C03641=1096.665,388.790,405.608,178.895,21.471,152.910
C03642=1096.660,388.542,405.645,178.892,21.465,152.909
C03643=1096.654,388.296,405.683,178.889,21.458,152.908
C03644=1096.648,388.049,405.721,178.886,21.452,152.907
C03645=1096.642,387.801,405.758,178.884,21.446,152.906
C03646=1096.637,387.555,405.796,178.881,21.440,152.905
C03647=1096.631,387.308,405.834,178.878,21.434,152.904
C03648=1096.625,387.061,405.871,178.876,21.428,152.903
C03649=1096.619,386.814,405.908,178.873,21.422,152.902
C03650=1096.614,386.567,405.945,178.869,21.416,152.901
C03651=1096.608,386.320,405.983,178.867,21.410,152.900
C03652=1096.601,386.072,406.021,178.864,21.404,152.899
C03653=1096.595,385.825,406.058,178.861,21.398,152.898
C03654=1096.590,385.579,406.094,178.859,21.392,152.897
C03655=1096.583,385.331,406.132,178.856,21.387,152.896
C03656=1096.578,385.084,406.170,178.853,21.381,152.895
C03657=1096.573,384.837,406.206,178.851,21.375,152.894
C03658=1096.567,384.590,406.244,178.847,21.369,152.893
C03659=1096.561,384.378,406.276,178.845,21.364,152.892
C03660=1096.556,384.167,406.308,178.843,21.359,152.891
C03661=1096.552,383.955,406.339,178.840,21.354,152.890
C03662=1096.546,383.743,406.371,178.838,21.349,152.890
C03663=1096.541,383.532,406.403,178.836,21.344,152.889
C03664=1096.536,383.321,406.435,178.833,21.339,152.888
C03665=1096.532,383.109,406.467,178.831,21.334,152.887
C03666=1096.527,382.897,406.499,178.828,21.329,152.886
C03667=1096.521,382.650,406.535,178.826,21.324,152.885
C03668=1096.515,382.403,406.572,178.823,21.318,152.885
C03669=1096.510,382.156,406.610,178.819,21.312,152.884
C03670=1096.503,381.909,406.646,178.816,21.306,152.883
C03671=1096.498,381.662,406.683,178.814,21.301,152.882
C03672=1096.492,381.414,406.720,178.811,21.295,152.881
C03673=1096.486,381.167,406.757,178.808,21.289,152.880
C03674=1096.480,380.920,406.794,178.805,21.284,152.879
C03675=1096.473,380.674,406.831,178.802,21.279,152.878
C03676=1096.468,380.426,406.868,178.799,21.273,152.877
C03677=1096.462,380.179,406.905,178.797,21.267,152.876
C03678=1096.456,379.932,406.942,178.794,21.262,152.876
C03679=1096.450,379.684,406.979,178.791,21.256,152.875
C03680=1096.445,379.438,407.015,178.788,21.251,152.874
C03681=1096.439,379.191,407.052,178.785,21.246,152.873
C03682=1096.433,378.944,407.088,178.782,21.240,152.872
C03683=1096.427,378.696,407.125,178.780,21.234,152.871
C03684=1096.421,378.449,407.162,178.777,21.229,152.870
C03685=1096.415,378.202,407.199,178.774,21.223,152.870
C03686=1096.410,377.955,407.236,178.771,21.218,152.869
C03687=1096.404,377.708,407.271,178.768,21.213,152.868
C03688=1096.398,377.460,407.308,178.765,21.207,152.867
C03689=1096.392,377.213,407.345,178.762,21.202,152.866
C03690=1096.387,376.966,407.382,178.759,21.196,152.865
C03691=1096.380,376.719,407.418,178.756,21.191,152.865
C03692=1096.375,376.472,407.455,178.754,21.186,152.864
C03693=1096.369,376.224,407.491,178.751,21.181,152.863
C03694=1096.364,375.977,407.528,178.748,21.176,152.862
C03695=1096.357,375.730,407.564,178.746,21.170,152.861
C03696=1096.352,375.483,407.601,178.743,21.165,152.860
C03697=1096.346,375.236,407.636,178.740,21.159,152.860
C03698=1096.341,374.988,407.673,178.737,21.154,152.859
C03699=1096.334,374.741,407.710,178.734,21.149,152.858
C03700=1096.329,374.494,407.745,178.731,21.144,152.857
C03701=1096.323,374.247,407.782,178.728,21.138,152.856
C03702=1096.317,374.000,407.819,178.725,21.133,152.856
C03703=1096.311,373.752,407.854,178.722,21.128,152.855
C03704=1096.305,373.505,407.892,178.719,21.123,152.854
C03705=1096.300,373.258,407.927,178.717,21.118,152.853
C03706=1096.294,373.011,407.963,178.714,21.113,152.853
C03707=1096.288,372.763,407.999,178.711,21.108,152.852
C03708=1096.282,372.516,408.036,178.708,21.102,152.851
C03709=1096.276,372.269,408.071,178.705,21.098,152.850
C03710=1096.270,372.022,408.108,178.702,21.092,152.850
C03711=1096.264,371.774,408.144,178.699,21.087,152.849
C03712=1096.259,371.527,408.181,178.696,21.082,152.848
C03713=1096.253,371.280,408.216,178.693,21.078,152.847
C03714=1096.247,371.033,408.252,178.691,21.072,152.847
C03715=1096.237,370.636,408.310,178.686,21.064,152.845
C03716=1096.228,370.241,408.368,178.681,21.056,152.844
C03717=1096.218,369.845,408.425,178.676,21.048,152.843
C03718=1096.210,369.448,408.483,178.672,21.041,152.842
C03719=1096.204,369.201,408.518,178.669,21.036,152.841
C03720=1096.198,368.954,408.555,178.666,21.031,152.841
C03721=1096.192,368.707,408.590,178.663,21.026,152.840
C03722=1096.187,368.460,408.626,178.659,21.021,152.839
C03723=1096.181,368.212,408.661,178.656,21.016,152.838
C03724=1096.175,367.965,408.698,178.654,21.011,152.838
C03725=1096.170,367.718,408.734,178.651,21.007,152.837
C03726=1096.164,367.470,408.770,178.648,21.001,152.836
C03727=1096.158,367.223,408.805,178.645,20.997,152.836
C03728=1096.152,366.975,408.841,178.642,20.992,152.835
C03729=1096.146,366.728,408.876,178.640,20.987,152.834
C03730=1096.141,366.481,408.912,178.636,20.982,152.834
C03731=1096.134,366.234,408.948,178.633,20.977,152.833
C03732=1096.129,365.987,408.984,178.630,20.973,152.832
C03733=1096.123,365.739,409.019,178.627,20.967,152.832
C03734=1096.118,365.492,409.055,178.625,20.963,152.831
C03735=1096.111,365.244,409.090,178.622,20.958,152.830
C03736=1096.105,364.997,409.126,178.619,20.953,152.830
C03737=1096.100,364.750,409.161,178.615,20.949,152.829
C03738=1096.094,364.502,409.197,178.612,20.944,152.828
C03739=1096.089,364.255,409.232,178.610,20.939,152.828
C03740=1096.083,364.007,409.268,178.607,20.935,152.827
C03741=1096.077,363.760,409.303,178.603,20.930,152.827
C03742=1096.071,363.512,409.339,178.600,20.925,152.826
C03743=1096.065,363.266,409.373,178.598,20.921,152.825
C03744=1096.059,363.018,409.409,178.595,20.916,152.825
C03745=1096.053,362.770,409.445,178.592,20.912,152.824
C03746=1096.048,362.523,409.480,178.588,20.907,152.824
C03747=1096.042,362.275,409.515,178.586,20.903,152.823
C03748=1096.037,362.028,409.551,178.583,20.898,152.822
C03749=1096.031,361.780,409.586,178.580,20.893,152.822
C03750=1096.024,361.534,409.621,178.577,20.889,152.821
C03751=1096.019,361.285,409.656,178.574,20.885,152.821
C03752=1096.013,361.038,409.691,178.571,20.880,152.820
C03753=1096.008,360.791,409.727,178.567,20.875,152.819
C03754=1096.002,360.544,409.763,178.565,20.871,152.819
C03755=1095.996,360.296,409.797,178.562,20.866,152.818
C03756=1095.990,360.049,409.832,178.559,20.862,152.818
C03757=1095.985,359.801,409.867,178.556,20.858,152.817
C03758=1095.979,359.553,409.903,178.553,20.853,152.817
C03759=1095.973,359.307,409.937,178.550,20.848,152.816
C03760=1095.967,359.059,409.973,178.546,20.844,152.815
C03761=1095.961,358.812,410.008,178.544,20.840,152.815
C03762=1095.955,358.564,410.042,178.541,20.835,152.814
C03763=1095.950,358.317,410.078,178.537,20.831,152.814
C03764=1095.944,358.069,410.112,178.535,20.827,152.813
C03765=1095.938,357.822,410.147,178.532,20.822,152.813
C03766=1095.933,357.574,410.182,178.528,20.818,152.812
C03767=1095.923,357.194,410.236,178.524,20.811,152.811
C03768=1095.914,356.813,410.290,178.520,20.804,152.810
C03769=1095.906,356.432,410.344,178.515,20.798,152.810
C03770=1095.897,356.051,410.397,178.511,20.791,152.809
C03771=1095.891,355.803,410.432,178.507,20.787,152.808
C03772=1095.885,355.556,410.466,178.504,20.782,152.808
C03773=1095.880,355.309,410.501,178.501,20.779,152.807
C03774=1095.873,355.061,410.536,178.498,20.774,152.807
C03775=1095.868,354.814,410.571,178.495,20.769,152.806
C03776=1095.862,354.566,410.605,178.492,20.765,152.806
C03777=1095.856,354.318,410.640,178.489,20.761,152.805
C03778=1095.851,354.071,410.675,178.487,20.757,152.805
C03779=1095.845,353.824,410.709,178.483,20.753,152.804
C03780=1095.839,353.576,410.744,178.480,20.748,152.804
C03781=1095.833,353.328,410.778,178.477,20.745,152.803
C03782=1095.828,353.081,410.813,178.474,20.740,152.803
C03783=1095.822,352.833,410.847,178.471,20.736,152.802
C03784=1095.816,352.586,410.882,178.468,20.732,152.802
C03785=1095.810,352.338,410.917,178.465,20.728,152.801
C03786=1095.805,352.091,410.951,178.462,20.724,152.801
C03787=1095.798,351.843,410.985,178.459,20.720,152.800
C03788=1095.793,351.596,411.020,178.455,20.715,152.800
C03789=1095.787,351.348,411.054,178.453,20.711,152.799
C03790=1095.781,351.100,411.089,178.450,20.707,152.799
C03791=1095.776,350.853,411.123,178.447,20.704,152.798
C03792=1095.770,350.605,411.157,178.443,20.699,152.798
C03793=1095.765,350.358,411.192,178.440,20.695,152.797
C03794=1095.758,350.110,411.226,178.438,20.691,152.797
C03795=1095.752,349.863,411.260,178.434,20.687,152.797
C03796=1095.747,349.615,411.295,178.432,20.683,152.796
C03797=1095.741,349.368,411.329,178.428,20.679,152.796
C03798=1095.735,349.120,411.363,178.425,20.675,152.795
C03799=1095.730,348.872,411.398,178.422,20.671,152.795
C03800=1095.724,348.625,411.432,178.420,20.667,152.794
C03801=1095.718,348.377,411.466,178.416,20.663,152.794
C03802=1095.712,348.130,411.500,178.413,20.659,152.793
C03803=1095.707,347.881,411.535,178.410,20.655,152.793
C03804=1095.701,347.634,411.569,178.407,20.651,152.793
C03805=1095.695,347.387,411.603,178.404,20.647,152.792
C03806=1095.689,347.140,411.637,178.401,20.643,152.792
C03807=1095.684,346.891,411.671,178.398,20.639,152.791
C03808=1095.678,346.644,411.705,178.395,20.635,152.791
C03809=1095.672,346.396,411.739,178.392,20.631,152.790
C03810=1095.666,346.148,411.772,178.389,20.627,152.790
C03811=1095.661,345.901,411.807,178.386,20.624,152.790
C03812=1095.655,345.654,411.841,178.382,20.619,152.789
C03813=1095.650,345.406,411.875,178.380,20.616,152.789
C03814=1095.644,345.158,411.909,178.376,20.612,152.788
C03815=1095.638,344.911,411.943,178.373,20.608,152.788
C03816=1095.633,344.663,411.976,178.370,20.604,152.788
C03817=1095.626,344.415,412.010,178.367,20.600,152.787
C03818=1095.620,344.168,412.044,178.364,20.596,152.787
C03819=1095.612,343.789,412.096,178.359,20.590,152.786
C03820=1095.603,343.411,412.147,178.355,20.584,152.786
C03821=1095.594,343.032,412.199,178.350,20.579,152.785
C03822=1095.586,342.654,412.250,178.346,20.574,152.784
C03823=1095.580,342.406,412.285,178.342,20.569,152.784
C03824=1095.574,342.158,412.318,178.340,20.566,152.784
C03825=1095.568,341.911,412.352,178.336,20.562,152.783
C03826=1095.563,341.663,412.385,178.333,20.558,152.783
C03827=1095.557,341.416,412.419,178.330,20.554,152.783
C03828=1095.551,341.168,412.452,178.327,20.551,152.782
C03829=1095.545,340.920,412.485,178.323,20.547,152.782
C03830=1095.539,340.673,412.519,178.321,20.544,152.782
C03831=1095.534,340.425,412.553,178.317,20.540,152.781
C03832=1095.528,340.177,412.586,178.314,20.536,152.781
C03833=1095.522,339.930,412.620,178.311,20.532,152.780
C03834=1095.517,339.682,412.654,178.308,20.529,152.780
C03835=1095.511,339.434,412.687,178.306,20.525,152.780
C03836=1095.505,339.187,412.721,178.302,20.521,152.779
C03837=1095.500,338.939,412.754,178.300,20.517,152.779
C03838=1095.494,338.691,412.788,178.296,20.514,152.779
C03839=1095.486,338.352,412.833,178.292,20.509,152.778
C03840=1095.479,338.012,412.879,178.287,20.504,152.778
C03841=1095.469,337.673,412.925,178.283,20.499,152.777
C03842=1095.462,337.333,412.971,178.279,20.494,152.777
C03843=1095.456,337.085,413.004,178.276,20.491,152.776
C03844=1095.450,336.838,413.037,178.273,20.487,152.776
C03845=1095.445,336.590,413.070,178.270,20.484,152.776
C03846=1095.439,336.342,413.104,178.266,20.480,152.776
C03847=1095.434,336.095,413.137,178.264,20.476,152.775
C03848=1095.428,335.847,413.169,178.261,20.473,152.775
C03849=1095.422,335.599,413.203,178.257,20.469,152.775
C03850=1095.417,335.351,413.236,178.254,20.466,152.774
C03851=1095.410,335.104,413.269,178.251,20.462,152.774
C03852=1095.405,334.856,413.302,178.248,20.459,152.774
C03853=1095.399,334.608,413.335,178.245,20.455,152.773
C03854=1095.394,334.360,413.369,178.242,20.451,152.773
C03855=1095.387,334.112,413.402,178.239,20.448,152.773
C03856=1095.382,333.864,413.435,178.236,20.445,152.772
C03857=1095.376,333.617,413.468,178.233,20.441,152.772
C03858=1095.371,333.370,413.501,178.230,20.438,152.772
C03859=1095.365,333.122,413.534,178.226,20.434,152.772
C03860=1095.359,332.874,413.567,178.223,20.431,152.771
C03861=1095.353,332.626,413.599,178.221,20.427,152.771
C03862=1095.348,332.378,413.633,178.217,20.424,152.771
C03863=1095.342,332.130,413.665,178.214,20.421,152.770
C03864=1095.336,331.882,413.699,178.211,20.417,152.770
C03865=1095.330,331.635,413.731,178.208,20.414,152.770
C03866=1095.325,331.387,413.764,178.205,20.411,152.770
C03867=1095.319,331.139,413.796,178.202,20.407,152.769
C03868=1095.313,330.891,413.830,178.198,20.404,152.769
C03869=1095.307,330.644,413.863,178.195,20.401,152.769
C03870=1095.301,330.396,413.895,178.193,20.397,152.769
C03871=1095.295,330.104,413.934,178.189,20.394,152.768
C03872=1095.287,329.811,413.973,178.184,20.389,152.768
C03873=1095.281,329.518,414.011,178.181,20.385,152.768
C03874=1095.273,329.226,414.049,178.177,20.381,152.767
C03875=1095.268,328.978,414.083,178.175,20.378,152.767
C03876=1095.262,328.729,414.115,178.172,20.375,152.767
C03877=1095.256,328.483,414.147,178.168,20.371,152.767
C03878=1095.251,328.234,414.180,178.165,20.368,152.767
C03879=1095.245,327.986,414.212,178.162,20.365,152.766
C03880=1095.238,327.739,414.245,178.158,20.361,152.766
C03881=1095.233,327.490,414.278,178.156,20.358,152.766
C03882=1095.227,327.243,414.310,178.153,20.355,152.766
C03883=1095.221,326.995,414.342,178.150,20.352,152.765
C03884=1095.216,326.747,414.375,178.146,20.348,152.765
C03885=1095.210,326.499,414.407,178.143,20.345,152.765
C03886=1095.204,326.252,414.440,178.140,20.342,152.765
C03887=1095.199,326.004,414.472,178.137,20.339,152.764
C03888=1095.193,325.755,414.505,178.134,20.336,152.764
C03889=1095.187,325.508,414.537,178.131,20.333,152.764
C03890=1095.181,325.260,414.569,178.128,20.329,152.764
C03891=1095.176,325.012,414.602,178.124,20.326,152.763
C03892=1095.170,324.764,414.634,178.121,20.323,152.763
C03893=1095.164,324.517,414.666,178.118,20.320,152.763
C03894=1095.158,324.269,414.699,178.115,20.316,152.763
C03895=1095.153,324.021,414.731,178.112,20.313,152.763
C03896=1095.147,323.773,414.763,178.109,20.310,152.762
C03897=1095.141,323.525,414.796,178.106,20.307,152.762
C03898=1095.135,323.277,414.828,178.102,20.304,152.762
C03899=1095.130,323.030,414.859,178.099,20.301,152.762
C03900=1095.125,322.781,414.892,178.096,20.298,152.762
C03901=1095.118,322.534,414.925,178.094,20.295,152.761
C03902=1095.113,322.286,414.956,178.090,20.291,152.761
C03903=1095.107,322.038,414.988,178.087,20.288,152.761
C03904=1095.101,321.790,415.020,178.084,20.285,152.761
C03905=1095.096,321.543,415.053,178.081,20.282,152.761
C03906=1095.090,321.294,415.085,178.078,20.279,152.760
C03907=1095.085,321.047,415.117,178.074,20.275,152.760
C03908=1095.079,320.799,415.149,178.071,20.272,152.760
C03909=1095.073,320.551,415.181,178.069,20.269,152.760
C03910=1095.067,320.303,415.213,178.066,20.266,152.759
C03911=1095.063,320.055,415.245,178.062,20.263,152.759
C03912=1095.057,319.807,415.277,178.059,20.260,152.759
C03913=1095.051,319.559,415.309,178.056,20.257,152.759
C03914=1095.045,319.311,415.341,178.053,20.254,152.759
C03915=1095.039,319.063,415.373,178.050,20.251,152.758
C03916=1095.034,318.815,415.405,178.046,20.247,152.758
C03917=1095.028,318.567,415.437,178.044,20.244,152.758
C03918=1095.022,318.320,415.468,178.041,20.241,152.758
C03919=1095.016,318.071,415.500,178.038,20.238,152.758
C03920=1095.011,317.824,415.532,178.034,20.235,152.757
C03921=1095.006,317.575,415.565,178.031,20.232,152.757
C03922=1095.000,317.328,415.596,178.028,20.229,152.757
C03923=1094.992,316.937,415.646,178.023,20.224,152.757
C03924=1094.982,316.546,415.696,178.018,20.219,152.757
C03925=1094.973,316.154,415.746,178.013,20.214,152.756
C03926=1094.965,315.762,415.796,178.009,20.210,152.756
C03927=1094.959,315.515,415.828,178.005,20.206,152.756
C03928=1094.954,315.267,415.860,178.002,20.203,152.756
C03929=1094.948,315.019,415.892,177.999,20.201,152.755
C03930=1094.942,314.770,415.923,177.996,20.198,152.755
C03931=1094.936,314.523,415.954,177.993,20.195,152.755
C03932=1094.930,314.275,415.986,177.990,20.192,152.755
C03933=1094.925,314.027,416.018,177.986,20.189,152.755
C03934=1094.919,313.779,416.049,177.983,20.186,152.755
C03935=1094.913,313.531,416.080,177.980,20.183,152.755
C03936=1094.907,313.283,416.112,177.977,20.180,152.754
C03937=1094.902,313.036,416.144,177.974,20.178,152.754
C03938=1094.896,312.788,416.174,177.971,20.175,152.754
C03939=1094.890,312.540,416.206,177.968,20.172,152.754
C03940=1094.884,312.292,416.238,177.964,20.169,152.754
C03941=1094.878,312.044,416.269,177.961,20.166,152.754
C03942=1094.873,311.796,416.300,177.958,20.163,152.754
C03943=1094.867,311.547,416.332,177.955,20.161,152.754
C03944=1094.861,311.300,416.363,177.952,20.158,152.754
C03945=1094.856,311.052,416.394,177.949,20.155,152.753
C03946=1094.849,310.804,416.425,177.946,20.152,152.753
C03947=1094.844,310.557,416.457,177.942,20.149,152.753
C03948=1094.838,310.308,416.488,177.939,20.146,152.753
C03949=1094.832,310.061,416.519,177.936,20.143,152.753
C03950=1094.827,309.812,416.550,177.933,20.141,152.753
C03951=1094.821,309.564,416.582,177.930,20.138,152.753
C03952=1094.815,309.316,416.612,177.927,20.135,152.753
C03953=1094.810,309.069,416.644,177.924,20.132,152.752
C03954=1094.803,308.820,416.675,177.920,20.129,152.752
C03955=1094.798,308.572,416.706,177.917,20.126,152.752
C03956=1094.792,308.325,416.737,177.914,20.124,152.752
C03957=1094.786,308.076,416.768,177.911,20.121,152.752
C03958=1094.780,307.829,416.799,177.908,20.118,152.752
C03959=1094.775,307.581,416.830,177.905,20.116,152.752
C03960=1094.770,307.333,416.861,177.902,20.113,152.752
C03961=1094.763,307.085,416.893,177.899,20.110,152.752
C03962=1094.758,306.837,416.923,177.896,20.107,152.751
C03963=1094.752,306.589,416.954,177.892,20.104,152.751
C03964=1094.747,306.341,416.986,177.889,20.101,152.751
C03965=1094.741,306.093,417.016,177.886,20.099,152.751
C03966=1094.735,305.845,417.047,177.883,20.096,152.751
C03967=1094.730,305.597,417.078,177.880,20.093,152.751
C03968=1094.724,305.349,417.109,177.876,20.091,152.751
C03969=1094.718,305.101,417.140,177.873,20.088,152.751
C03970=1094.713,304.853,417.171,177.870,20.085,152.751
C03971=1094.707,304.605,417.201,177.867,20.082,152.751
C03972=1094.701,304.357,417.232,177.863,20.079,152.751
C03973=1094.696,304.110,417.263,177.860,20.076,152.750
C03974=1094.690,303.862,417.294,177.857,20.074,152.750
C03975=1094.681,303.472,417.342,177.853,20.070,152.750
C03976=1094.672,303.083,417.390,177.847,20.065,152.750
C03977=1094.664,302.695,417.439,177.843,20.061,152.750
C03978=1094.655,302.306,417.487,177.838,20.057,152.750
C03979=1094.649,302.058,417.517,177.835,20.054,152.750
C03980=1094.644,301.810,417.548,177.831,20.051,152.750
C03981=1094.638,301.562,417.578,177.828,20.048,152.749
C03982=1094.632,301.315,417.609,177.825,20.045,152.749
C03983=1094.627,301.067,417.640,177.822,20.043,152.749
C03984=1094.621,300.819,417.670,177.819,20.040,152.749
C03985=1094.616,300.570,417.701,177.816,20.038,152.749
C03986=1094.610,300.322,417.732,177.813,20.035,152.749
C03987=1094.604,300.074,417.762,177.810,20.032,152.749
C03988=1094.599,299.826,417.793,177.806,20.030,152.749
C03989=1094.593,299.578,417.823,177.803,20.027,152.749
C03990=1094.588,299.330,417.853,177.800,20.024,152.749
C03991=1094.582,299.082,417.884,177.797,20.021,152.748
C03992=1094.577,298.834,417.914,177.794,20.019,152.748
C03993=1094.571,298.586,417.945,177.791,20.016,152.748
C03994=1094.566,298.338,417.976,177.788,20.014,152.748
C03995=1094.560,298.090,418.006,177.785,20.011,152.748
C03996=1094.554,297.842,418.036,177.782,20.008,152.748
C03997=1094.549,297.594,418.066,177.779,20.006,152.748
C03998=1094.543,297.346,418.096,177.775,20.003,152.748
C03999=1094.538,297.098,418.127,177.771,20.000,152.748
C04000=1094.532,296.849,418.157,177.768,19.998,152.748
C04001=1094.526,296.602,418.187,177.765,19.995,152.748
C04002=1094.521,296.354,418.218,177.762,19.992,152.748
C04003=1094.515,296.105,418.247,177.759,19.990,152.748
C04004=1094.509,295.858,418.277,177.756,19.987,152.748
C04005=1094.503,295.610,418.308,177.753,19.985,152.748
C04006=1094.498,295.361,418.337,177.750,19.982,152.748
C04007=1094.492,295.113,418.368,177.746,19.980,152.748
C04008=1094.486,294.865,418.399,177.743,19.977,152.748
C04009=1094.480,294.616,418.428,177.740,19.974,152.747
C04010=1094.474,294.369,418.459,177.737,19.972,152.747
C04011=1094.469,294.121,418.489,177.734,19.969,152.747
C04012=1094.463,293.872,418.519,177.731,19.967,152.747
C04013=1094.457,293.625,418.549,177.727,19.964,152.747
C04014=1094.452,293.376,418.579,177.724,19.962,152.747
C04015=1094.446,293.128,418.609,177.721,19.959,152.747
C04016=1094.441,292.881,418.638,177.718,19.957,152.747
C04017=1094.435,292.633,418.668,177.715,19.954,152.747
C04018=1094.430,292.384,418.698,177.712,19.952,152.747
C04019=1094.424,292.137,418.728,177.709,19.949,152.747
C04020=1094.418,291.888,418.758,177.706,19.946,152.747
C04021=1094.412,291.640,418.788,177.702,19.944,152.747
C04022=1094.407,291.392,418.818,177.699,19.942,152.747
C04023=1094.401,291.143,418.848,177.696,19.939,152.747
C04024=1094.396,290.896,418.878,177.693,19.937,152.747
C04025=1094.390,290.647,418.908,177.690,19.934,152.747
C04026=1094.385,290.399,418.937,177.687,19.931,152.747
C04027=1094.376,290.025,418.982,177.682,19.928,152.747
C04028=1094.367,289.650,419.028,177.677,19.924,152.747
C04029=1094.359,289.275,419.072,177.673,19.921,152.747
C04030=1094.350,288.900,419.117,177.668,19.917,152.747
C04031=1094.344,288.652,419.146,177.665,19.915,152.747
C04032=1094.339,288.404,419.176,177.662,19.912,152.747
C04033=1094.333,288.156,419.206,177.659,19.910,152.747
C04034=1094.327,287.908,419.235,177.656,19.907,152.747
C04035=1094.321,287.659,419.265,177.652,19.905,152.747
C04036=1094.316,287.411,419.295,177.649,19.903,152.747
C04037=1094.310,287.162,419.324,177.646,19.900,152.747
C04038=1094.304,286.915,419.354,177.643,19.898,152.747
C04039=1094.299,286.667,419.383,177.639,19.895,152.747
C04040=1094.293,286.419,419.413,177.636,19.893,152.747
C04041=1094.287,286.170,419.442,177.633,19.890,152.747
C04042=1094.281,285.922,419.472,177.630,19.888,152.747
C04043=1094.276,285.674,419.501,177.627,19.886,152.747
C04044=1094.271,285.426,419.531,177.624,19.883,152.747
C04045=1094.265,285.178,419.560,177.620,19.880,152.747
C04046=1094.259,284.929,419.589,177.617,19.878,152.747
C04047=1094.254,284.681,419.619,177.615,19.876,152.747
C04048=1094.247,284.433,419.648,177.612,19.874,152.747
C04049=1094.243,284.185,419.677,177.608,19.872,152.747
C04050=1094.237,283.937,419.707,177.605,19.869,152.747
C04051=1094.231,283.688,419.736,177.602,19.866,152.747
C04052=1094.225,283.440,419.765,177.599,19.864,152.747
C04053=1094.220,283.191,419.795,177.596,19.862,152.747
C04054=1094.214,282.944,419.824,177.593,19.859,152.747
C04055=1094.209,282.696,419.853,177.589,19.857,152.747
C04056=1094.202,282.447,419.882,177.586,19.854,152.747
C04057=1094.197,282.199,419.912,177.583,19.852,152.747
C04058=1094.192,281.951,419.941,177.580,19.850,152.747
C04059=1094.186,281.703,419.970,177.576,19.847,152.747
C04060=1094.180,281.455,420.000,177.574,19.845,152.747
C04061=1094.175,281.207,420.028,177.571,19.843,152.747
C04062=1094.169,280.958,420.058,177.568,19.840,152.747
C04063=1094.163,280.710,420.087,177.564,19.838,152.747
C04064=1094.158,280.462,420.116,177.561,19.836,152.747
C04065=1094.152,280.214,420.145,177.558,19.833,152.747
C04066=1094.147,279.965,420.174,177.555,19.831,152.747
C04067=1094.140,279.717,420.203,177.551,19.829,152.747
C04068=1094.135,279.469,420.233,177.548,19.826,152.747
C04069=1094.129,279.221,420.261,177.546,19.825,152.747
C04070=1094.123,278.972,420.290,177.543,19.822,152.747
C04071=1094.118,278.724,420.319,177.539,19.820,152.747
C04072=1094.112,278.477,420.348,177.536,19.817,152.747
C04073=1094.107,278.227,420.377,177.533,19.815,152.747
C04074=1094.101,277.979,420.406,177.530,19.813,152.747
C04075=1094.096,277.732,420.435,177.526,19.810,152.747
C04076=1094.090,277.483,420.463,177.523,19.808,152.747
C04077=1094.084,277.235,420.492,177.520,19.806,152.747
C04078=1094.079,276.986,420.521,177.518,19.804,152.747
C04079=1094.070,276.621,420.564,177.513,19.800,152.747
C04080=1094.062,276.255,420.607,177.508,19.797,152.747
C04081=1094.054,275.890,420.648,177.504,19.794,152.747
C04082=1094.045,275.525,420.691,177.499,19.790,152.747
C04083=1094.040,275.277,420.719,177.496,19.788,152.747
C04084=1094.034,275.028,420.748,177.493,19.785,152.747
C04085=1094.028,274.780,420.777,177.489,19.783,152.747
C04086=1094.023,274.532,420.806,177.486,19.781,152.747
C04087=1094.017,274.283,420.834,177.484,19.779,152.747
C04088=1094.011,274.036,420.863,177.480,19.777,152.747
C04089=1094.005,273.787,420.891,177.477,19.774,152.747
C04090=1094.000,273.538,420.920,177.474,19.772,152.747
C04091=1093.995,273.291,420.949,177.470,19.770,152.748
C04092=1093.989,273.042,420.977,177.467,19.767,152.747
C04093=1093.983,272.794,421.006,177.464,19.765,152.748
C04094=1093.977,272.546,421.034,177.462,19.763,152.747
C04095=1093.972,272.297,421.063,177.458,19.761,152.748
C04096=1093.966,272.049,421.092,177.455,19.759,152.748
C04097=1093.960,271.800,421.120,177.452,19.756,152.748
C04098=1093.955,271.552,421.148,177.449,19.754,152.748
C04099=1093.949,271.304,421.176,177.445,19.752,152.748
C04100=1093.943,271.056,421.205,177.443,19.750,152.748
C04101=1093.938,270.807,421.234,177.440,19.748,152.748
C04102=1093.933,270.559,421.262,177.436,19.745,152.748
C04103=1093.927,270.310,421.290,177.433,19.743,152.748
C04104=1093.921,270.063,421.319,177.430,19.741,152.748
C04105=1093.915,269.814,421.347,177.427,19.739,152.748
C04106=1093.910,269.566,421.375,177.424,19.737,152.748
C04107=1093.904,269.317,421.404,177.421,19.735,152.748
C04108=1093.899,269.069,421.432,177.418,19.732,152.748
C04109=1093.893,268.820,421.460,177.414,19.730,152.748
C04110=1093.887,268.573,421.489,177.411,19.728,152.748
C04111=1093.881,268.324,421.517,177.408,19.726,152.748
C04112=1093.876,268.076,421.545,177.405,19.724,152.748
C04113=1093.870,267.828,421.573,177.402,19.722,152.748
C04114=1093.864,267.579,421.601,177.399,19.720,152.749
C04115=1093.859,267.331,421.629,177.395,19.717,152.749
C04116=1093.853,267.083,421.657,177.393,19.715,152.749
C04117=1093.847,266.834,421.686,177.390,19.713,152.749
C04118=1093.842,266.586,421.714,177.386,19.711,152.749
C04119=1093.836,266.337,421.742,177.383,19.709,152.749
C04120=1093.831,266.089,421.770,177.380,19.706,152.749
C04121=1093.825,265.840,421.798,177.377,19.705,152.749
C04122=1093.819,265.592,421.826,177.374,19.702,152.749
C04123=1093.814,265.344,421.854,177.371,19.700,152.749
C04124=1093.808,265.095,421.883,177.367,19.698,152.749
C04125=1093.803,264.847,421.910,177.364,19.695,152.749
C04126=1093.797,264.599,421.939,177.362,19.694,152.749
C04127=1093.791,264.351,421.967,177.358,19.692,152.749
C04128=1093.785,264.102,421.995,177.355,19.690,152.749
C04129=1093.780,263.853,422.022,177.352,19.687,152.749
C04130=1093.774,263.605,422.050,177.348,19.685,152.750
C04131=1093.765,263.242,422.090,177.344,19.682,152.750
C04132=1093.757,262.880,422.132,177.339,19.679,152.750
C04133=1093.748,262.517,422.172,177.335,19.676,152.750
C04134=1093.740,262.155,422.213,177.330,19.673,152.750
C04135=1093.734,261.906,422.240,177.328,19.672,152.750
C04136=1093.729,261.658,422.268,177.324,19.669,152.750
C04137=1093.723,261.409,422.296,177.321,19.667,152.750
C04138=1093.717,261.162,422.323,177.318,19.665,152.750
C04139=1093.711,260.912,422.351,177.315,19.663,152.750
C04140=1093.706,260.664,422.379,177.312,19.661,152.750
C04141=1093.700,260.417,422.406,177.309,19.659,152.751
C04142=1093.694,260.167,422.434,177.305,19.657,152.751
C04143=1093.689,259.919,422.462,177.303,19.655,152.751
C04144=1093.683,259.671,422.489,177.299,19.653,152.751
C04145=1093.677,259.422,422.517,177.296,19.651,152.751
C04146=1093.672,259.174,422.545,177.293,19.649,152.751
C04147=1093.665,258.926,422.573,177.290,19.647,152.751
C04148=1093.660,258.677,422.600,177.287,19.645,152.751
C04149=1093.655,258.429,422.628,177.284,19.642,152.751
C04150=1093.649,258.180,422.654,177.280,19.640,152.751
C04151=1093.643,257.932,422.683,177.278,19.639,152.751
C04152=1093.637,257.683,422.709,177.275,19.637,152.751
C04153=1093.632,257.435,422.737,177.271,19.634,152.752
C04154=1093.626,257.186,422.765,177.268,19.632,152.752
C04155=1093.620,256.938,422.792,177.265,19.631,152.752
C04156=1093.615,256.689,422.820,177.262,19.628,152.752
C04157=1093.609,256.441,422.847,177.259,19.626,152.752
C04158=1093.604,256.192,422.874,177.256,19.624,152.752
C04159=1093.597,255.945,422.902,177.253,19.622,152.752
C04160=1093.592,255.696,422.929,177.250,19.620,152.752
C04161=1093.587,255.447,422.957,177.246,19.618,152.752
C04162=1093.581,255.199,422.984,177.244,19.616,152.752
C04163=1093.576,254.950,423.011,177.241,19.614,152.752
C04164=1093.570,254.702,423.039,177.237,19.612,152.753
C04165=1093.565,254.454,423.066,177.234,19.610,152.753
C04166=1093.558,254.205,423.093,177.232,19.608,152.753
C04167=1093.553,253.957,423.121,177.228,19.606,152.753
C04168=1093.547,253.708,423.148,177.225,19.604,152.753
C04169=1093.542,253.460,423.175,177.221,19.602,152.753
C04170=1093.536,253.212,423.202,177.219,19.600,152.753
C04171=1093.530,252.963,423.230,177.216,19.598,152.753
C04172=1093.525,252.714,423.256,177.212,19.596,152.753
C04173=1093.520,252.465,423.284,177.210,19.594,152.753
C04174=1093.513,252.218,423.311,177.207,19.592,152.753
C04175=1093.508,251.969,423.338,177.203,19.589,152.753
C04176=1093.503,251.721,423.365,177.200,19.587,152.754
C04177=1093.498,251.472,423.392,177.197,19.586,152.754
C04178=1093.491,251.223,423.419,177.194,19.584,152.754
C04179=1093.486,250.975,423.447,177.191,19.581,152.754
C04180=1093.480,250.727,423.474,177.188,19.580,152.754
C04181=1093.475,250.478,423.501,177.185,19.577,152.754
C04182=1093.469,250.230,423.528,177.182,19.575,152.754
C04183=1093.461,249.864,423.568,177.178,19.572,152.754
C04184=1093.453,249.499,423.607,177.173,19.569,152.754
C04185=1093.445,249.133,423.647,177.168,19.567,152.754
C04186=1093.437,248.768,423.686,177.164,19.564,152.755
C04187=1093.431,248.519,423.713,177.161,19.561,152.755
C04188=1093.426,248.270,423.740,177.158,19.559,152.755
C04189=1093.420,248.022,423.767,177.154,19.557,152.755
C04190=1093.415,247.773,423.794,177.152,19.556,152.755
C04191=1093.409,247.524,423.821,177.149,19.553,152.755
C04192=1093.403,247.276,423.848,177.145,19.551,152.755
C04193=1093.398,247.027,423.875,177.143,19.550,152.755
C04194=1093.392,246.779,423.902,177.139,19.548,152.755
C04195=1093.387,246.531,423.928,177.136,19.545,152.755
C04196=1093.381,246.282,423.955,177.133,19.544,152.755
C04197=1093.376,246.034,423.982,177.130,19.542,152.756
C04198=1093.370,245.785,424.009,177.127,19.540,152.756
C04199=1093.365,245.536,424.035,177.124,19.538,152.756
C04200=1093.359,245.288,424.061,177.121,19.536,152.756
C04201=1093.353,245.040,424.088,177.118,19.534,152.756
C04202=1093.348,244.791,424.115,177.115,19.532,152.756
C04203=1093.342,244.543,424.142,177.112,19.530,152.756
C04204=1093.336,244.294,424.168,177.108,19.528,152.756
C04205=1093.331,244.045,424.194,177.106,19.526,152.756
C04206=1093.325,243.797,424.221,177.103,19.524,152.756
C04207=1093.319,243.549,424.248,177.099,19.522,152.756
C04208=1093.314,243.300,424.275,177.097,19.520,152.757
C04209=1093.309,243.051,424.301,177.094,19.518,152.757
C04210=1093.303,242.803,424.328,177.091,19.516,152.757
C04211=1093.297,242.554,424.354,177.087,19.515,152.757
C04212=1093.292,242.306,424.381,177.084,19.512,152.757
C04213=1093.286,242.057,424.407,177.082,19.511,152.757
C04214=1093.280,241.808,424.433,177.078,19.509,152.757
C04215=1093.275,241.560,424.460,177.075,19.507,152.757
C04216=1093.269,241.311,424.486,177.072,19.505,152.758
C04217=1093.263,241.063,424.513,177.069,19.503,152.758
C04218=1093.258,240.814,424.539,177.066,19.501,152.758
C04219=1093.252,240.565,424.565,177.063,19.499,152.758
C04220=1093.246,240.317,424.592,177.060,19.497,152.758
C04221=1093.241,240.068,424.618,177.057,19.495,152.758
C04222=1093.235,239.820,424.644,177.054,19.493,152.758
C04223=1093.229,239.571,424.671,177.051,19.491,152.758
C04224=1093.224,239.322,424.697,177.048,19.490,152.758
C04225=1093.218,239.074,424.724,177.045,19.487,152.758
C04226=1093.213,238.825,424.750,177.041,19.486,152.759
C04227=1093.207,238.578,424.775,177.039,19.484,152.759
C04228=1093.201,238.329,424.801,177.035,19.482,152.759
C04229=1093.195,238.080,424.828,177.033,19.480,152.759
C04230=1093.190,237.831,424.854,177.029,19.478,152.759
C04231=1093.184,237.583,424.880,177.026,19.476,152.759
C04232=1093.179,237.334,424.906,177.024,19.475,152.759
C04233=1093.173,237.086,424.933,177.020,19.472,152.759
C04234=1093.168,236.837,424.959,177.017,19.470,152.760
C04235=1093.159,236.465,424.998,177.013,19.468,152.760
C04236=1093.150,236.092,425.037,177.009,19.465,152.760
C04237=1093.143,235.719,425.076,177.004,19.462,152.760
C04238=1093.134,235.347,425.114,176.999,19.459,152.760
C04239=1093.128,235.099,425.141,176.996,19.457,152.760
C04240=1093.123,234.850,425.167,176.994,19.455,152.760
C04241=1093.117,234.601,425.193,176.990,19.454,152.761
C04242=1093.112,234.352,425.219,176.987,19.452,152.761
C04243=1093.106,234.105,425.245,176.984,19.450,152.761
C04244=1093.101,233.856,425.270,176.981,19.448,152.761
C04245=1093.095,233.607,425.296,176.978,19.446,152.761
C04246=1093.090,233.358,425.322,176.975,19.444,152.761
C04247=1093.083,233.110,425.348,176.972,19.443,152.761
C04248=1093.078,232.861,425.374,176.969,19.441,152.761
C04249=1093.073,232.613,425.400,176.966,19.438,152.762
C04250=1093.067,232.364,425.426,176.963,19.437,152.762
C04251=1093.061,232.116,425.452,176.960,19.435,152.762
C04252=1093.055,231.867,425.478,176.957,19.433,152.762
C04253=1093.050,231.618,425.503,176.954,19.431,152.762
C04254=1093.045,231.369,425.529,176.951,19.430,152.762
C04255=1093.039,231.121,425.555,176.948,19.428,152.762
C04256=1093.033,230.872,425.581,176.945,19.426,152.762
C04257=1093.028,230.623,425.606,176.942,19.424,152.763
C04258=1093.022,230.375,425.631,176.939,19.422,152.763
C04259=1093.017,230.126,425.657,176.936,19.420,152.763
C04260=1093.010,229.878,425.683,176.933,19.418,152.763
C04261=1093.005,229.629,425.709,176.930,19.417,152.763
C04262=1092.999,229.381,425.734,176.927,19.415,152.763
C04263=1092.994,229.132,425.760,176.923,19.413,152.763
C04264=1092.988,228.883,425.786,176.921,19.411,152.763
C04265=1092.983,228.635,425.811,176.917,19.409,152.764
C04266=1092.977,228.386,425.837,176.915,19.407,152.764
C04267=1092.971,228.137,425.862,176.912,19.405,152.764
C04268=1092.966,227.888,425.888,176.909,19.404,152.764
C04269=1092.960,227.640,425.913,176.906,19.402,152.764
C04270=1092.954,227.391,425.939,176.903,19.400,152.764
C04271=1092.949,227.142,425.964,176.900,19.398,152.764
C04272=1092.944,226.894,425.990,176.897,19.397,152.764
C04273=1092.937,226.645,426.015,176.894,19.395,152.765
C04274=1092.932,226.396,426.041,176.890,19.393,152.765
C04275=1092.926,226.148,426.066,176.888,19.391,152.765
C04276=1092.921,225.899,426.092,176.884,19.389,152.765
C04277=1092.915,225.650,426.117,176.882,19.388,152.765
C04278=1092.910,225.402,426.143,176.879,19.385,152.765
C04279=1092.904,225.153,426.167,176.876,19.384,152.765
C04280=1092.898,224.904,426.193,176.873,19.382,152.765
C04281=1092.893,224.656,426.218,176.870,19.381,152.766
C04282=1092.887,224.407,426.243,176.867,19.379,152.766
C04283=1092.881,224.158,426.269,176.864,19.377,152.766
C04284=1092.876,223.910,426.294,176.861,19.375,152.766
C04285=1092.870,223.661,426.320,176.858,19.373,152.766
C04286=1092.865,223.413,426.345,176.855,19.371,152.766
C04287=1092.856,223.031,426.383,176.851,19.368,152.766
C04288=1092.848,222.650,426.422,176.846,19.365,152.767
C04289=1092.839,222.269,426.460,176.841,19.363,152.767
C04290=1092.831,221.888,426.499,176.837,19.360,152.767
C04291=1092.825,221.639,426.524,176.834,19.358,152.767
C04292=1092.819,221.391,426.549,176.831,19.357,152.767
C04293=1092.814,221.142,426.574,176.828,19.355,152.768
C04294=1092.808,220.893,426.600,176.825,19.353,152.768
C04295=1092.802,220.645,426.624,176.822,19.351,152.768
C04296=1092.796,220.396,426.649,176.819,19.350,152.768
C04297=1092.791,220.148,426.675,176.816,19.348,152.768
C04298=1092.785,219.898,426.699,176.813,19.346,152.768
C04299=1092.780,219.650,426.724,176.810,19.344,152.768
C04300=1092.774,219.401,426.749,176.807,19.343,152.768
C04301=1092.768,219.152,426.774,176.804,19.341,152.769
C04302=1092.763,218.903,426.799,176.801,19.339,152.769
C04303=1092.757,218.655,426.824,176.798,19.337,152.769
C04304=1092.752,218.406,426.849,176.795,19.336,152.769
C04305=1092.746,218.158,426.874,176.792,19.334,152.769
C04306=1092.740,217.909,426.898,176.790,19.332,152.769
C04307=1092.735,217.660,426.924,176.786,19.330,152.769
C04308=1092.729,217.411,426.948,176.784,19.328,152.769
C04309=1092.723,217.163,426.974,176.780,19.327,152.770
C04310=1092.718,216.914,426.998,176.778,19.325,152.770
C04311=1092.712,216.665,427.023,176.774,19.323,152.770
C04312=1092.706,216.417,427.048,176.772,19.321,152.770
C04313=1092.701,216.168,427.072,176.768,19.319,152.770
C04314=1092.696,215.919,427.098,176.766,19.318,152.770
C04315=1092.690,215.671,427.122,176.762,19.316,152.771
C04316=1092.684,215.421,427.147,176.760,19.314,152.771
C04317=1092.679,215.173,427.172,176.756,19.312,152.771
C04318=1092.673,214.924,427.196,176.754,19.311,152.771
C04319=1092.668,214.676,427.221,176.751,19.309,152.771
C04320=1092.661,214.427,427.246,176.748,19.307,152.771
C04321=1092.656,214.178,427.270,176.745,19.306,152.771
C04322=1092.652,213.929,427.295,176.742,19.304,152.771
C04323=1092.646,213.680,427.320,176.739,19.302,152.772
C04324=1092.640,213.432,427.345,176.736,19.300,152.772
C04325=1092.634,213.183,427.369,176.734,19.298,152.772
C04326=1092.629,212.934,427.393,176.730,19.296,152.772
C04327=1092.624,212.686,427.418,176.728,19.295,152.772
C04328=1092.618,212.436,427.442,176.724,19.293,152.772
C04329=1092.612,212.188,427.467,176.722,19.291,152.772
C04330=1092.606,211.939,427.492,176.718,19.289,152.773
C04331=1092.601,211.691,427.516,176.716,19.288,152.773
C04332=1092.596,211.442,427.540,176.713,19.287,152.773
C04333=1092.589,211.193,427.565,176.710,19.284,152.773
C04334=1092.584,210.944,427.589,176.707,19.283,152.773
C04335=1092.578,210.695,427.613,176.704,19.281,152.773
C04336=1092.572,210.447,427.638,176.701,19.279,152.773
C04337=1092.567,210.199,427.663,176.698,19.277,152.774
C04338=1092.561,209.949,427.687,176.695,19.276,152.774
C04339=1092.553,209.572,427.724,176.691,19.273,152.774
C04340=1092.545,209.194,427.761,176.687,19.271,152.774
C04341=1092.535,208.818,427.798,176.682,19.268,152.774
C04342=1092.527,208.441,427.834,176.677,19.265,152.775
C04343=1092.504,207.422,427.933,176.617,19.237,152.779
C04344=1092.499,207.173,427.957,176.614,19.236,152.780
C04345=1092.493,206.925,427.980,176.611,19.235,152.780
C04346=1092.488,206.676,428.004,176.608,19.235,152.780
C04347=1092.482,206.426,428.029,176.605,19.234,152.781
C04348=1092.476,206.178,428.052,176.601,19.232,152.781
C04349=1092.471,205.929,428.076,176.598,19.232,152.781
C04350=1092.465,205.681,428.100,176.595,19.231,152.782
C04351=1092.460,205.432,428.124,176.592,19.230,152.782
C04352=1092.454,205.182,428.148,176.589,19.229,152.782
C04353=1092.448,204.934,428.171,176.586,19.229,152.783
C04354=1092.443,204.685,428.196,176.583,19.228,152.783
C04355=1092.438,204.436,428.219,176.580,19.227,152.783
C04356=1092.432,204.188,428.243,176.577,19.226,152.784
C04357=1092.426,203.939,428.267,176.574,19.225,152.784
C04358=1092.421,203.690,428.290,176.571,19.224,152.785
C04359=1092.415,203.441,428.315,176.568,19.223,152.785
C04360=1092.409,203.192,428.338,176.565,19.223,152.785
C04361=1092.404,202.944,428.362,176.562,19.222,152.786
C04362=1092.399,202.694,428.385,176.559,19.221,152.786
C04363=1092.393,202.446,428.409,176.555,19.220,152.786
C04364=1092.387,202.197,428.432,176.552,19.219,152.787
C04365=1092.382,201.949,428.456,176.549,19.219,152.787
C04366=1092.375,201.699,428.480,176.547,19.218,152.787
C04367=1092.370,201.450,428.504,176.544,19.217,152.788
C04368=1092.364,201.201,428.527,176.541,19.216,152.788
C04369=1092.358,200.953,428.550,176.538,19.216,152.789
C04370=1092.353,200.704,428.574,176.535,19.215,152.789
C04371=1092.347,200.456,428.598,176.532,19.214,152.789
C04372=1092.341,200.207,428.621,176.529,19.213,152.790
C04373=1092.336,199.958,428.645,176.525,19.212,152.790
C04374=1092.330,199.709,428.668,176.522,19.211,152.790
C04375=1092.324,199.460,428.692,176.519,19.210,152.791
C04376=1092.319,199.211,428.715,176.516,19.210,152.791
C04377=1092.313,198.962,428.738,176.513,19.209,152.791
C04378=1092.307,198.714,428.762,176.510,19.208,152.792
C04379=1092.302,198.465,428.785,176.508,19.207,152.792
C04380=1092.296,198.216,428.808,176.505,19.207,152.793
C04381=1092.290,197.968,428.832,176.502,19.206,152.793
C04382=1092.285,197.718,428.856,176.499,19.205,152.793
C04383=1092.279,197.469,428.879,176.495,19.204,152.794
C04384=1092.273,197.221,428.902,176.492,19.203,152.794
C04385=1092.268,196.971,428.926,176.489,19.203,152.794
C04386=1092.262,196.722,428.949,176.486,19.201,152.795
C04387=1092.256,196.473,428.972,176.483,19.201,152.795
C04388=1092.250,196.225,428.996,176.480,19.200,152.795
C04389=1092.245,195.976,429.019,176.478,19.199,152.796
C04390=1092.240,195.727,429.042,176.475,19.198,152.796
C04391=1092.234,195.478,429.065,176.472,19.198,152.796
C04392=1092.229,195.230,429.089,176.469,19.197,152.797
C04393=1092.223,194.981,429.112,176.466,19.196,152.797
C04394=1092.217,194.732,429.135,176.463,19.195,152.798
C04395=1092.211,194.483,429.158,176.460,19.194,152.798
C04396=1092.206,194.234,429.182,176.456,19.193,152.798
C04397=1092.201,193.985,429.205,176.453,19.192,152.798
C04398=1092.195,193.737,429.228,176.450,19.191,152.799
C04399=1092.190,193.488,429.251,176.447,19.191,152.799
C04400=1092.185,193.239,429.274,176.445,19.190,152.799
C04401=1092.179,192.990,429.297,176.442,19.189,152.800
C04402=1092.173,192.741,429.320,176.439,19.188,152.800
C04403=1092.167,192.492,429.343,176.436,19.187,152.801
C04404=1092.161,192.216,429.369,176.433,19.187,152.801
C04405=1092.155,191.940,429.395,176.429,19.185,152.801
C04406=1092.149,191.664,429.421,176.426,19.184,152.802
C04407=1092.143,191.389,429.445,176.423,19.184,152.802
C04408=1092.138,191.139,429.469,176.420,19.182,152.802
C04409=1092.132,190.890,429.492,176.417,19.181,152.803
C04410=1092.126,190.642,429.515,176.414,19.181,152.803
C04411=1092.120,190.393,429.538,176.411,19.180,152.803
C04412=1092.115,190.144,429.561,176.408,19.179,152.804
C04413=1092.110,189.895,429.584,176.405,19.178,152.804
C04414=1092.104,189.646,429.607,176.402,19.177,152.804
C04415=1092.099,189.397,429.630,176.399,19.176,152.805
C04416=1092.093,189.149,429.653,176.396,19.176,152.805
C04417=1092.087,188.900,429.676,176.394,19.175,152.805
C04418=1092.082,188.651,429.699,176.391,19.174,152.806
C04419=1092.076,188.402,429.722,176.388,19.173,152.806
C04420=1092.071,188.152,429.744,176.385,19.172,152.806
C04421=1092.065,187.903,429.767,176.382,19.171,152.807
C04422=1092.060,187.655,429.790,176.379,19.170,152.807
C04423=1092.055,187.406,429.813,176.376,19.169,152.807
C04424=1092.049,187.157,429.836,176.374,19.168,152.808
C04425=1092.043,186.908,429.859,176.371,19.168,152.808
C04426=1092.037,186.659,429.882,176.368,19.167,152.808
C04427=1092.033,186.411,429.904,176.365,19.166,152.809
C04428=1092.027,186.162,429.927,176.362,19.165,152.809
C04429=1092.022,185.912,429.950,176.359,19.164,152.809
C04430=1092.016,185.664,429.973,176.356,19.163,152.809
C04431=1092.011,185.415,429.995,176.354,19.162,152.810
C04432=1092.006,185.166,430.018,176.351,19.161,152.810
C04433=1092.000,184.917,430.041,176.348,19.160,152.810
C04434=1091.993,184.668,430.063,176.345,19.160,152.811
C04435=1091.988,184.419,430.085,176.342,19.159,152.811
C04436=1091.982,184.170,430.108,176.339,19.158,152.811
C04437=1091.977,183.921,430.131,176.336,19.157,152.812
C04438=1091.971,183.673,430.154,176.333,19.157,152.812
C04439=1091.965,183.424,430.176,176.330,19.156,152.812
C04440=1091.959,183.175,430.198,176.327,19.155,152.813
C04441=1091.954,182.926,430.221,176.325,19.154,152.813
C04442=1091.948,182.676,430.244,176.322,19.153,152.814
C04443=1091.942,182.428,430.266,176.319,19.152,152.814
C04444=1091.936,182.179,430.289,176.316,19.151,152.814
C04445=1091.931,181.930,430.311,176.313,19.151,152.815
C04446=1091.925,181.681,430.333,176.310,19.150,152.815
C04447=1091.919,181.432,430.355,176.307,19.149,152.815
C04448=1091.914,181.183,430.378,176.304,19.148,152.816
C04449=1091.908,180.934,430.401,176.301,19.147,152.816
C04450=1091.902,180.686,430.423,176.299,19.146,152.816
C04451=1091.897,180.437,430.445,176.296,19.146,152.817
C04452=1091.891,180.187,430.468,176.293,19.145,152.817
C04453=1091.885,179.939,430.490,176.290,19.144,152.817
C04454=1091.879,179.689,430.512,176.287,19.143,152.817
C04455=1091.874,179.441,430.535,176.284,19.142,152.818
C04456=1091.868,179.192,430.557,176.281,19.141,152.818
C04457=1091.862,178.943,430.579,176.278,19.140,152.819
C04458=1091.857,178.693,430.602,176.276,19.139,152.819
C04459=1091.851,178.445,430.624,176.273,19.139,152.819
C04460=1091.846,178.196,430.646,176.270,19.138,152.819
C04461=1091.840,177.947,430.669,176.267,19.137,152.820
C04462=1091.834,177.699,430.690,176.264,19.136,152.820
C04463=1091.829,177.450,430.713,176.261,19.135,152.820
C04464=1091.823,177.200,430.735,176.258,19.134,152.821
C04465=1091.817,176.951,430.757,176.256,19.133,152.821
C04466=1091.812,176.703,430.780,176.253,19.133,152.821
C04467=1091.806,176.453,430.802,176.250,19.131,152.822
C04468=1091.800,176.177,430.826,176.247,19.131,152.822
C04469=1091.794,175.900,430.850,176.244,19.130,152.822
C04470=1091.788,175.624,430.875,176.240,19.129,152.823
C04471=1091.781,175.347,430.900,176.237,19.127,152.823
C04472=1091.775,175.099,430.922,176.234,19.127,152.823
C04473=1091.770,174.850,430.944,176.232,19.126,152.824
C04474=1091.765,174.600,430.966,176.229,19.125,152.824
C04475=1091.759,174.353,430.988,176.226,19.124,152.824
C04476=1091.753,174.103,431.010,176.223,19.123,152.825
C04477=1091.747,173.854,431.032,176.221,19.122,152.825
C04478=1091.742,173.605,431.054,176.218,19.122,152.825
C04479=1091.737,173.356,431.077,176.215,19.121,152.826
C04480=1091.731,173.107,431.099,176.213,19.120,152.826
C04481=1091.726,172.858,431.120,176.210,19.119,152.826
C04482=1091.720,172.609,431.142,176.207,19.118,152.826
C04483=1091.714,172.361,431.165,176.204,19.117,152.827
C04484=1091.708,172.112,431.186,176.201,19.116,152.827
C04485=1091.703,171.862,431.209,176.198,19.115,152.827
C04486=1091.697,171.614,431.230,176.196,19.114,152.828
C04487=1091.692,171.364,431.252,176.193,19.113,152.828
C04488=1091.687,171.115,431.274,176.190,19.112,152.828
C04489=1091.681,170.867,431.296,176.187,19.111,152.829
C04490=1091.676,170.618,431.318,176.184,19.110,152.829
C04491=1091.670,170.369,431.340,176.182,19.109,152.829
C04492=1091.664,170.119,431.362,176.179,19.108,152.829
C04493=1091.659,169.871,431.383,176.177,19.108,152.830
C04494=1091.653,169.621,431.405,176.174,19.107,152.830
C04495=1091.648,169.373,431.427,176.171,19.106,152.830
C04496=1091.642,169.123,431.449,176.168,19.105,152.831
C04497=1091.637,168.875,431.470,176.165,19.104,152.831
C04498=1091.631,168.625,431.492,176.163,19.103,152.831
C04499=1091.626,168.376,431.514,176.160,19.102,152.831
C04500=1091.620,168.127,431.536,176.157,19.101,152.832
C04501=1091.615,167.878,431.557,176.154,19.099,152.832
C04502=1091.609,167.629,431.579,176.151,19.099,152.832
C04503=1091.604,167.380,431.601,176.149,19.098,152.833
C04504=1091.598,167.131,431.623,176.146,19.097,152.833
C04505=1091.593,166.882,431.644,176.144,19.096,152.833
C04506=1091.586,166.633,431.666,176.141,19.095,152.833
C04507=1091.582,166.384,431.688,176.138,19.094,152.834
C04508=1091.576,166.136,431.709,176.136,19.093,152.834
C04509=1091.571,165.886,431.731,176.133,19.092,152.834
C04510=1091.565,165.638,431.752,176.130,19.091,152.834
C04511=1091.560,165.388,431.775,176.127,19.090,152.835
C04512=1091.554,165.140,431.796,176.124,19.089,152.835
C04513=1091.549,164.890,431.818,176.122,19.088,152.835
C04514=1091.543,164.642,431.839,176.119,19.087,152.836
C04515=1091.538,164.393,431.860,176.116,19.086,152.836
C04516=1091.532,164.143,431.882,176.114,19.085,152.836
C04517=1091.527,163.895,431.904,176.111,19.084,152.836
C04518=1091.521,163.645,431.926,176.109,19.083,152.837
C04519=1091.516,163.397,431.947,176.106,19.082,152.837
C04520=1091.510,163.148,431.968,176.103,19.081,152.837
C04521=1091.505,162.898,431.990,176.100,19.080,152.837
C04522=1091.500,162.650,432.011,176.098,19.078,152.838
C04523=1091.495,162.401,432.033,176.095,19.077,152.838
C04524=1091.489,162.152,432.055,176.092,19.076,152.838
C04525=1091.483,161.902,432.075,176.090,19.076,152.838
C04526=1091.478,161.653,432.097,176.087,19.075,152.839
C04527=1091.472,161.404,432.119,176.084,19.074,152.839
C04528=1091.467,161.156,432.140,176.082,19.073,152.839
C04529=1091.461,160.906,432.161,176.079,19.072,152.839
C04530=1091.455,160.658,432.182,176.076,19.071,152.840
C04531=1091.449,160.408,432.204,176.073,19.070,152.840
C04532=1091.443,160.132,432.227,176.071,19.068,152.840
C04533=1091.438,159.855,432.251,176.068,19.068,152.841
C04534=1091.431,159.578,432.275,176.065,19.067,152.841
C04535=1091.425,159.302,432.299,176.062,19.066,152.841
C04536=1091.419,159.052,432.320,176.059,19.065,152.841
C04537=1091.414,158.803,432.341,176.057,19.064,152.842
C04538=1091.408,158.554,432.361,176.054,19.062,152.842
C04539=1091.402,158.305,432.383,176.051,19.061,152.842
C04540=1091.397,158.057,432.404,176.048,19.060,152.843
C04541=1091.391,157.807,432.425,176.045,19.060,152.843
C04542=1091.386,157.558,432.447,176.043,19.059,152.843
C04543=1091.381,157.309,432.468,176.041,19.058,152.843
C04544=1091.375,157.060,432.489,176.038,19.057,152.844
C04545=1091.369,156.811,432.511,176.035,19.056,152.844
C04546=1091.364,156.562,432.531,176.032,19.055,152.844
C04547=1091.358,156.313,432.552,176.030,19.054,152.844
C04548=1091.352,156.064,432.573,176.027,19.053,152.845
C04549=1091.347,155.815,432.595,176.024,19.051,152.845
C04550=1091.342,155.566,432.615,176.022,19.051,152.845
C04551=1091.335,155.317,432.637,176.019,19.050,152.845
C04552=1091.330,155.068,432.657,176.017,19.049,152.846
C04553=1091.325,154.819,432.679,176.014,19.048,152.846
C04554=1091.319,154.569,432.700,176.011,19.046,152.846
C04555=1091.313,154.321,432.721,176.008,19.045,152.847
C04556=1091.308,154.072,432.741,176.006,19.045,152.847
C04557=1091.302,153.822,432.762,176.004,19.044,152.847
C04558=1091.296,153.573,432.784,176.001,19.043,152.847
C04559=1091.291,153.324,432.804,175.998,19.042,152.848
C04560=1091.285,153.075,432.826,175.995,19.040,152.848
C04561=1091.280,152.826,432.846,175.993,19.039,152.848
C04562=1091.275,152.577,432.867,175.991,19.039,152.848
C04563=1091.269,152.328,432.888,175.988,19.038,152.849
C04564=1091.262,152.079,432.908,175.985,19.036,152.849
C04565=1091.257,151.830,432.929,175.983,19.035,152.849
C04566=1091.252,151.581,432.950,175.980,19.034,152.849
C04567=1091.246,151.332,432.971,175.977,19.033,152.849
C04568=1091.240,151.082,432.992,175.975,19.032,152.850
C04569=1091.235,150.834,433.013,175.973,19.031,152.850
C04570=1091.230,150.585,433.034,175.970,19.030,152.850
C04571=1091.224,150.335,433.054,175.967,19.029,152.850
C04572=1091.218,150.086,433.076,175.964,19.028,152.851
C04573=1091.212,149.837,433.096,175.961,19.027,152.851
C04574=1091.207,149.588,433.116,175.960,19.026,152.851
C04575=1091.202,149.339,433.137,175.957,19.025,152.851
C04576=1091.196,149.090,433.158,175.954,19.024,152.852
C04577=1091.190,148.841,433.179,175.952,19.023,152.852
C04578=1091.185,148.592,433.200,175.949,19.021,152.852
C04579=1091.179,148.343,433.220,175.947,19.021,152.852
C04580=1091.173,148.094,433.241,175.944,19.020,152.853
C04581=1091.168,147.845,433.262,175.941,19.019,152.853
C04582=1091.162,147.595,433.282,175.939,19.018,152.853
C04583=1091.156,147.347,433.302,175.936,19.017,152.853
C04584=1091.151,147.097,433.323,175.933,19.015,152.854
C04585=1091.145,146.848,433.344,175.931,19.014,152.854
C04586=1091.140,146.599,433.365,175.929,19.013,152.854
C04587=1091.134,146.350,433.385,175.926,19.012,152.854
C04588=1091.128,146.101,433.405,175.923,19.011,152.855
C04589=1091.123,145.852,433.426,175.920,19.010,152.855
C04590=1091.117,145.603,433.446,175.918,19.009,152.855
C04591=1091.111,145.353,433.467,175.916,19.008,152.855
C04592=1091.106,145.104,433.487,175.913,19.007,152.855
C04593=1091.100,144.856,433.507,175.910,19.006,152.856
C04594=1091.095,144.606,433.528,175.908,19.005,152.856
C04595=1091.090,144.357,433.549,175.906,19.004,152.856
C04596=1091.082,144.080,433.572,175.903,19.003,152.856
C04597=1091.077,143.803,433.595,175.899,19.001,152.857
C04598=1091.071,143.526,433.617,175.897,19.000,152.857
C04599=1091.064,143.250,433.640,175.894,18.999,152.857
C04600=1091.059,143.001,433.660,175.891,18.998,152.857
C04601=1091.054,142.751,433.681,175.889,18.997,152.858
C04602=1091.048,142.503,433.701,175.887,18.996,152.858
C04603=1091.042,142.253,433.722,175.884,18.994,152.858
C04604=1091.036,142.004,433.742,175.881,18.993,152.858
C04605=1091.030,141.755,433.762,175.879,18.993,152.859
C04606=1091.025,141.506,433.783,175.877,18.991,152.859
C04607=1091.019,141.256,433.802,175.874,18.990,152.859
C04608=1091.014,141.007,433.822,175.871,18.989,152.859
C04609=1091.009,140.758,433.843,175.869,18.988,152.859
C04610=1091.003,140.509,433.863,175.867,18.987,152.860
C04611=1090.998,140.260,433.883,175.864,18.986,152.860
C04612=1090.992,140.011,433.903,175.861,18.985,152.860
C04613=1090.986,139.762,433.924,175.859,18.983,152.860
C04614=1090.980,139.513,433.944,175.857,18.983,152.860
C04615=1090.975,139.264,433.965,175.854,18.981,152.861
C04616=1090.969,139.014,433.984,175.852,18.980,152.861
C04617=1090.964,138.765,434.005,175.849,18.979,152.861
C04618=1090.958,138.516,434.025,175.846,18.978,152.861
C04619=1090.952,138.267,434.045,175.844,18.977,152.862
C04620=1090.946,138.018,434.065,175.842,18.976,152.862
C04621=1090.941,137.768,434.085,175.839,18.974,152.862
C04622=1090.935,137.520,434.105,175.836,18.973,152.862
C04623=1090.930,137.271,434.126,175.835,18.972,152.862
C04624=1090.924,137.022,434.145,175.832,18.971,152.863
C04625=1090.919,136.772,434.165,175.829,18.970,152.863
C04626=1090.913,136.523,434.185,175.827,18.969,152.863
C04627=1090.907,136.274,434.205,175.825,18.968,152.863
C04628=1090.902,136.025,434.226,175.822,18.967,152.863
C04629=1090.896,135.776,434.245,175.819,18.965,152.864
C04630=1090.891,135.527,434.266,175.817,18.964,152.864
C04631=1090.885,135.278,434.286,175.815,18.964,152.864
C04632=1090.879,135.028,434.305,175.812,18.962,152.864
C04633=1090.874,134.779,434.325,175.809,18.961,152.864
C04634=1090.868,134.531,434.345,175.807,18.960,152.865
C04635=1090.863,134.281,434.365,175.805,18.959,152.865
C04636=1090.857,134.032,434.385,175.802,18.958,152.865
C04637=1090.851,133.783,434.405,175.800,18.956,152.865
C04638=1090.846,133.533,434.425,175.797,18.955,152.866
C04639=1090.840,133.285,434.445,175.795,18.954,152.866
C04640=1090.834,133.036,434.465,175.793,18.953,152.866
C04641=1090.829,132.786,434.485,175.790,18.952,152.866
C04642=1090.823,132.537,434.505,175.787,18.950,152.866
C04643=1090.818,132.287,434.524,175.785,18.950,152.866
C04644=1090.812,132.039,434.544,175.783,18.948,152.867
C04645=1090.807,131.789,434.564,175.780,18.947,152.867
C04646=1090.801,131.540,434.584,175.777,18.946,152.867
C04647=1090.795,131.292,434.604,175.776,18.945,152.867
C04648=1090.790,131.042,434.623,175.773,18.944,152.867
C04649=1090.784,130.793,434.643,175.770,18.942,152.868
C04650=1090.778,130.544,434.663,175.768,18.942,152.868
C04651=1090.772,130.295,434.683,175.766,18.941,152.868
C04652=1090.766,130.045,434.702,175.763,18.939,152.868
C04653=1090.760,129.797,434.722,175.760,18.938,152.869
C04654=1090.755,129.547,434.742,175.759,18.937,152.869
C04655=1090.749,129.298,434.762,175.756,18.936,152.869
C04656=1090.744,129.049,434.781,175.753,18.935,152.869
C04657=1090.738,128.799,434.800,175.752,18.934,152.869
C04658=1090.732,128.550,434.820,175.749,18.933,152.869
C04659=1090.726,128.301,434.839,175.746,18.931,152.870
C04660=1090.720,128.024,434.861,175.744,18.930,152.870
C04661=1090.714,127.747,434.884,175.741,18.929,152.870
C04662=1090.708,127.469,434.905,175.738,18.927,152.870
C04663=1090.701,127.193,434.927,175.736,18.926,152.870
C04664=1090.696,126.944,434.945,175.733,18.925,152.871
C04665=1090.691,126.695,434.966,175.731,18.924,152.871
C04666=1090.685,126.445,434.985,175.729,18.923,152.871
C04667=1090.679,126.196,435.005,175.726,18.921,152.871
C04668=1090.673,125.947,435.024,175.723,18.920,152.871
C04669=1090.668,125.698,435.044,175.722,18.919,152.871
C04670=1090.662,125.448,435.063,175.719,18.918,152.872
C04671=1090.656,125.200,435.083,175.716,18.916,152.872
C04672=1090.651,124.951,435.102,175.714,18.916,152.872
C04673=1090.645,124.701,435.121,175.712,18.914,152.872
C04674=1090.639,124.452,435.140,175.709,18.913,152.873
C04675=1090.633,124.203,435.160,175.707,18.912,152.873
C04676=1090.628,123.954,435.179,175.705,18.910,152.873
C04677=1090.623,123.704,435.199,175.702,18.909,152.873
C04678=1090.617,123.455,435.219,175.700,18.908,152.873
C04679=1090.612,123.206,435.238,175.698,18.907,152.873
C04680=1090.606,122.957,435.257,175.695,18.906,152.873
C04681=1090.600,122.708,435.277,175.693,18.904,152.874
C04682=1090.595,122.458,435.296,175.691,18.904,152.874
C04683=1090.589,122.209,435.315,175.688,18.902,152.874
C04684=1090.584,121.961,435.335,175.686,18.900,152.874
C04685=1090.578,121.711,435.354,175.683,18.899,152.874
C04686=1090.572,121.462,435.373,175.681,18.898,152.874
C04687=1090.566,121.212,435.392,175.679,18.897,152.875
C04688=1090.561,120.963,435.412,175.676,18.896,152.875
C04689=1090.556,120.714,435.431,175.674,18.895,152.875
C04690=1090.550,120.465,435.450,175.672,18.893,152.875
C04691=1090.544,120.216,435.470,175.669,18.892,152.875
C04692=1090.538,119.966,435.489,175.667,18.891,152.875
C04693=1090.533,119.718,435.508,175.665,18.889,152.876
C04694=1090.528,119.468,435.527,175.662,18.888,152.876
C04695=1090.522,119.219,435.546,175.661,18.887,152.876
C04696=1090.516,118.969,435.566,175.658,18.886,152.876
C04697=1090.511,118.721,435.584,175.655,18.884,152.876
C04698=1090.505,118.471,435.604,175.654,18.883,152.876
C04699=1090.500,118.222,435.623,175.651,18.882,152.877
C04700=1090.495,117.973,435.642,175.649,18.880,152.877
C04701=1090.489,117.724,435.661,175.647,18.879,152.877
C04702=1090.483,117.474,435.680,175.644,18.878,152.877
C04703=1090.478,117.225,435.700,175.642,18.877,152.877
C04704=1090.472,116.976,435.718,175.639,18.875,152.877
C04705=1090.467,116.727,435.738,175.637,18.874,152.877
C04706=1090.460,116.477,435.756,175.635,18.872,152.877
C04707=1090.455,116.229,435.775,175.632,18.871,152.878
C04708=1090.450,115.979,435.794,175.630,18.870,152.878
C04709=1090.444,115.730,435.814,175.628,18.869,152.878
C04710=1090.439,115.481,435.833,175.625,18.867,152.878
C04711=1090.433,115.232,435.852,175.624,18.866,152.878
C04712=1090.427,114.982,435.871,175.621,18.865,152.878
C04713=1090.422,114.734,435.890,175.619,18.863,152.879
C04714=1090.417,114.484,435.908,175.617,18.862,152.879
C04715=1090.411,114.234,435.928,175.614,18.861,152.879
C04716=1090.405,113.986,435.946,175.612,18.859,152.879
C04717=1090.400,113.736,435.965,175.610,18.858,152.879
C04718=1090.394,113.487,435.984,175.607,18.857,152.879
C04719=1090.389,113.238,436.003,175.605,18.856,152.879
C04720=1090.383,112.989,436.022,175.603,18.854,152.879
C04721=1090.377,112.739,436.041,175.601,18.853,152.880
C04722=1090.372,112.490,436.059,175.598,18.851,152.880
C04723=1090.366,112.241,436.079,175.596,18.851,152.880
C04724=1090.360,111.963,436.100,175.594,18.849,152.880
C04725=1090.354,111.687,436.120,175.591,18.848,152.880
C04726=1090.348,111.409,436.141,175.589,18.846,152.880
C04727=1090.341,111.132,436.162,175.586,18.844,152.880
C04728=1090.335,110.884,436.181,175.583,18.843,152.881
C04729=1090.329,110.634,436.200,175.582,18.842,152.881
C04730=1090.324,110.384,436.218,175.579,18.841,152.881
C04731=1090.318,110.136,436.237,175.577,18.839,152.881
C04732=1090.313,109.886,436.256,175.575,18.838,152.881
C04733=1090.307,109.637,436.275,175.572,18.837,152.881
C04734=1090.301,109.388,436.293,175.571,18.836,152.882
C04735=1090.296,109.138,436.312,175.568,18.834,152.882
C04736=1090.290,108.890,436.330,175.566,18.833,152.882
C04737=1090.284,108.640,436.349,175.564,18.832,152.882
C04738=1090.279,108.391,436.368,175.561,18.830,152.882
C04739=1090.273,108.142,436.386,175.559,18.829,152.882
C04740=1090.268,107.892,436.405,175.557,18.828,152.882
C04741=1090.262,107.644,436.423,175.555,18.827,152.882
C04742=1090.256,107.394,436.442,175.552,18.825,152.883
C04743=1090.250,107.144,436.460,175.550,18.824,152.883
C04744=1090.245,106.896,436.479,175.548,18.822,152.883
C04745=1090.239,106.646,436.498,175.546,18.821,152.883
C04746=1090.234,106.397,436.516,175.544,18.820,152.883
C04747=1090.228,106.148,436.535,175.541,18.818,152.883
C04748=1090.222,105.898,436.553,175.539,18.817,152.883
C04749=1090.217,105.649,436.572,175.537,18.816,152.883
C04750=1090.211,105.400,436.590,175.534,18.814,152.884
C04751=1090.206,105.151,436.609,175.533,18.813,152.884
C04752=1090.199,104.901,436.627,175.530,18.811,152.884
C04753=1090.194,104.652,436.646,175.528,18.810,152.884
C04754=1090.189,104.402,436.664,175.526,18.809,152.884
C04755=1090.183,104.154,436.682,175.524,18.807,152.884
C04756=1090.178,103.904,436.701,175.522,18.806,152.884
C04757=1090.172,103.655,436.719,175.519,18.805,152.884
C04758=1090.167,103.405,436.738,175.517,18.803,152.884
C04759=1090.161,103.157,436.756,175.515,18.802,152.885
C04760=1090.155,102.907,436.775,175.513,18.800,152.885
C04761=1090.150,102.658,436.793,175.510,18.799,152.885
C04762=1090.144,102.408,436.811,175.508,18.798,152.885
C04763=1090.138,102.160,436.830,175.506,18.796,152.885
C04764=1090.133,101.910,436.848,175.504,18.795,152.885
C04765=1090.127,101.662,436.866,175.502,18.794,152.885
C04766=1090.122,101.411,436.885,175.499,18.792,152.885
C04767=1090.116,101.162,436.903,175.498,18.791,152.885
C04768=1090.110,100.913,436.921,175.495,18.789,152.886
C04769=1090.105,100.664,436.939,175.493,18.788,152.886
C04770=1090.099,100.415,436.958,175.491,18.787,152.886
C04771=1090.093,100.166,436.976,175.488,18.785,152.886
C04772=1090.088,99.916,436.994,175.487,18.784,152.886
C04773=1090.082,99.667,437.012,175.484,18.783,152.886
C04774=1090.076,99.418,437.030,175.483,18.781,152.886
C04775=1090.071,99.168,437.049,175.480,18.780,152.886
C04776=1090.065,98.919,437.067,175.478,18.778,152.886
C04777=1090.059,98.670,437.085,175.476,18.777,152.887
C04778=1090.054,98.420,437.103,175.473,18.776,152.887
C04779=1090.048,98.172,437.122,175.472,18.775,152.887
C04780=1090.042,97.922,437.139,175.469,18.773,152.887
C04781=1090.036,97.673,437.157,175.467,18.771,152.887
C04782=1090.031,97.423,437.176,175.465,18.770,152.887
C04783=1090.025,97.174,437.194,175.463,18.768,152.887
C04784=1090.019,96.925,437.212,175.461,18.767,152.887
C04785=1090.014,96.675,437.230,175.459,18.766,152.887
C04786=1090.009,96.426,437.248,175.456,18.764,152.887
C04787=1090.002,96.177,437.266,175.454,18.763,152.888
C04788=1089.996,95.900,437.286,175.452,18.762,152.888
C04789=1089.991,95.623,437.306,175.449,18.760,152.888
C04790=1089.983,95.346,437.326,175.447,18.758,152.888
C04791=1089.977,95.069,437.346,175.445,18.756,152.888
C04792=1089.972,94.820,437.363,175.443,18.755,152.888
C04793=1089.966,94.570,437.383,175.440,18.754,152.888
C04794=1089.961,94.321,437.400,175.439,18.753,152.888
C04795=1089.954,94.071,437.418,175.436,18.751,152.888
C04796=1089.949,93.822,437.436,175.434,18.750,152.889
C04797=1089.944,93.573,437.454,175.432,18.748,152.888
C04798=1089.938,93.323,437.472,175.430,18.746,152.889
C04799=1089.933,93.074,437.489,175.428,18.745,152.889
C04800=1089.927,92.825,437.507,175.426,18.744,152.889
C04801=1089.921,92.576,437.526,175.423,18.742,152.889
C04802=1089.916,92.327,437.544,175.422,18.741,152.889
C04803=1089.910,92.078,437.561,175.419,18.739,152.889
C04804=1089.904,91.828,437.579,175.418,18.738,152.889
C04805=1089.899,91.579,437.597,175.415,18.736,152.889
C04806=1089.894,91.330,437.615,175.413,18.735,152.889
C04807=1089.888,91.080,437.633,175.411,18.733,152.889
C04808=1089.882,90.831,437.650,175.409,18.732,152.889
C04809=1089.876,90.581,437.668,175.407,18.731,152.890
C04810=1089.871,90.332,437.686,175.404,18.729,152.890
C04811=1089.865,90.083,437.703,175.403,18.728,152.890
C04812=1089.859,89.833,437.721,175.400,18.726,152.890
C04813=1089.853,89.584,437.739,175.399,18.725,152.890
C04814=1089.848,89.335,437.757,175.396,18.723,152.890
C04815=1089.842,89.085,437.774,175.394,18.722,152.890
C04816=1089.836,88.836,437.792,175.392,18.721,152.890
C04817=1089.831,88.587,437.810,175.390,18.719,152.890
C04818=1089.825,88.338,437.828,175.388,18.718,152.890
C04819=1089.819,88.088,437.845,175.386,18.716,152.890
C04820=1089.814,87.839,437.863,175.384,18.715,152.891
C04821=1089.807,87.590,437.881,175.381,18.713,152.891
C04822=1089.802,87.341,437.898,175.379,18.711,152.891
C04823=1089.797,87.091,437.915,175.378,18.710,152.891
C04824=1089.791,86.841,437.933,175.375,18.709,152.891
C04825=1089.785,86.592,437.950,175.373,18.708,152.891
C04826=1089.780,86.343,437.968,175.371,18.706,152.891
C04827=1089.773,86.093,437.986,175.369,18.705,152.891
C04828=1089.768,85.844,438.004,175.367,18.703,152.891
C04829=1089.762,85.595,438.021,175.365,18.702,152.891
C04830=1089.757,85.346,438.039,175.363,18.700,152.891
C04831=1089.751,85.096,438.056,175.361,18.698,152.891
C04832=1089.746,84.847,438.073,175.359,18.697,152.891
C04833=1089.740,84.598,438.091,175.357,18.695,152.891
C04834=1089.735,84.349,438.109,175.355,18.694,152.892
C04835=1089.728,84.099,438.126,175.352,18.693,152.892
C04836=1089.722,83.850,438.143,175.351,18.691,152.892
C04837=1089.717,83.601,438.160,175.348,18.689,152.892
C04838=1089.711,83.352,438.178,175.347,18.688,152.892
C04839=1089.705,83.102,438.196,175.345,18.686,152.892
C04840=1089.700,82.852,438.213,175.343,18.685,152.892
C04841=1089.695,82.603,438.230,175.340,18.684,152.892
C04842=1089.689,82.354,438.248,175.338,18.682,152.892
C04843=1089.683,82.104,438.266,175.336,18.681,152.892
C04844=1089.678,81.855,438.283,175.334,18.679,152.892
C04845=1089.672,81.606,438.300,175.333,18.677,152.892
C04846=1089.667,81.357,438.318,175.330,18.676,152.892
C04847=1089.661,81.107,438.334,175.329,18.674,152.892
C04848=1089.655,80.858,438.352,175.326,18.673,152.892
C04849=1089.649,80.609,438.370,175.324,18.672,152.893
C04850=1089.644,80.359,438.386,175.322,18.670,152.892
C04851=1089.638,80.110,438.404,175.320,18.669,152.893
C04852=1089.632,79.833,438.423,175.318,18.667,152.893
C04853=1089.626,79.556,438.443,175.316,18.665,152.893
C04854=1089.620,79.279,438.462,175.313,18.663,152.893
C04855=1089.613,79.001,438.481,175.311,18.661,152.893
C04856=1089.608,78.752,438.498,175.310,18.660,152.893
C04857=1089.602,78.503,438.516,175.307,18.658,152.893
C04858=1089.596,78.254,438.532,175.305,18.657,152.893
C04859=1089.591,78.005,438.549,175.303,18.655,152.893
C04860=1089.585,77.755,438.567,175.301,18.654,152.893
C04861=1089.579,77.506,438.584,175.299,18.652,152.893
C04862=1089.574,77.256,438.601,175.298,18.651,152.893
C04863=1089.568,77.007,438.618,175.295,18.649,152.893
C04864=1089.562,76.758,438.636,175.294,18.648,152.893
C04865=1089.556,76.508,438.652,175.291,18.646,152.893
C04866=1089.550,76.259,438.670,175.290,18.645,152.893
C04867=1089.545,76.009,438.687,175.287,18.643,152.893
C04868=1089.540,75.760,438.704,175.285,18.641,152.893
C04869=1089.534,75.511,438.721,175.283,18.640,152.894
C04870=1089.528,75.262,438.738,175.281,18.638,152.894
C04871=1089.523,75.012,438.755,175.279,18.637,152.894
C04872=1089.516,74.763,438.772,175.277,18.635,152.894
C04873=1089.511,74.513,438.789,175.275,18.634,152.894
C04874=1089.506,74.264,438.806,175.273,18.632,152.894
C04875=1089.499,74.015,438.823,175.271,18.631,152.894
C04876=1089.494,73.765,438.840,175.269,18.629,152.894
C04877=1089.488,73.516,438.857,175.268,18.627,152.894
C04878=1089.483,73.267,438.874,175.265,18.626,152.894
C04879=1089.477,73.018,438.891,175.264,18.624,152.894
C04880=1089.471,72.768,438.907,175.261,18.623,152.894
C04881=1089.466,72.519,438.924,175.260,18.621,152.894
C04882=1089.460,72.269,438.942,175.257,18.620,152.894
C04883=1089.454,72.020,438.958,175.256,18.618,152.894
C04884=1089.449,71.771,438.976,175.253,18.617,152.894
C04885=1089.443,71.521,438.992,175.252,18.615,152.894
C04886=1089.437,71.272,439.009,175.249,18.613,152.894
C04887=1089.432,71.023,439.027,175.248,18.612,152.894
C04888=1089.426,70.773,439.043,175.245,18.610,152.894
C04889=1089.421,70.524,439.060,175.244,18.609,152.894
C04890=1089.414,70.275,439.077,175.242,18.607,152.894
C04891=1089.409,70.025,439.094,175.240,18.606,152.894
C04892=1089.403,69.776,439.110,175.238,18.604,152.894
C04893=1089.398,69.526,439.127,175.236,18.602,152.895
C04894=1089.392,69.277,439.144,175.234,18.600,152.895
C04895=1089.387,69.028,439.161,175.232,18.599,152.895
C04896=1089.381,68.778,439.177,175.230,18.597,152.895
C04897=1089.375,68.529,439.194,175.228,18.596,152.895
C04898=1089.369,68.279,439.211,175.226,18.594,152.895
C04899=1089.363,68.030,439.228,175.224,18.593,152.895
C04900=1089.357,67.780,439.244,175.222,18.591,152.895
C04901=1089.352,67.531,439.261,175.221,18.589,152.895
C04902=1089.346,67.282,439.278,175.218,18.588,152.895
C04903=1089.341,67.032,439.295,175.217,18.586,152.895
C04904=1089.335,66.783,439.311,175.214,18.585,152.895
C04905=1089.330,66.533,439.328,175.213,18.583,152.895
C04906=1089.324,66.284,439.344,175.210,18.582,152.895
C04907=1089.318,66.035,439.362,175.209,18.580,152.895
C04908=1089.312,65.786,439.378,175.207,18.578,152.895
C04909=1089.306,65.536,439.394,175.205,18.577,152.895
C04910=1089.301,65.287,439.411,175.203,18.575,152.895
C04911=1089.295,65.037,439.427,175.201,18.574,152.895
C04912=1089.290,64.788,439.444,175.199,18.572,152.895
C04913=1089.284,64.538,439.460,175.197,18.570,152.895
C04914=1089.278,64.289,439.477,175.196,18.569,152.895
C04915=1089.272,64.040,439.494,175.194,18.567,152.895
C04916=1089.265,63.763,439.512,175.191,18.566,152.895
C04917=1089.260,63.486,439.530,175.190,18.564,152.895
C04918=1089.253,63.209,439.548,175.187,18.562,152.895
C04919=1089.246,62.932,439.567,175.185,18.560,152.895
C04920=1089.240,62.682,439.584,175.183,18.559,152.895
C04921=1089.234,62.433,439.600,175.181,18.557,152.895
C04922=1089.229,62.183,439.617,175.180,18.556,152.895
C04923=1089.223,61.934,439.633,175.177,18.554,152.896
C04924=1089.217,61.685,439.649,175.176,18.552,152.895
C04925=1089.211,61.435,439.665,175.173,18.550,152.895
C04926=1089.205,61.186,439.682,175.172,18.549,152.896
C04927=1089.200,60.936,439.699,175.169,18.547,152.896
C04928=1089.194,60.687,439.715,175.168,18.546,152.896
C04929=1089.188,60.438,439.731,175.166,18.544,152.896
C04930=1089.182,60.188,439.747,175.164,18.543,152.896
C04931=1089.176,59.939,439.764,175.162,18.541,152.896
C04932=1089.171,59.689,439.780,175.160,18.539,152.896
C04933=1089.165,59.440,439.797,175.159,18.538,152.896
C04934=1089.159,59.191,439.813,175.156,18.536,152.896
C04935=1089.153,58.941,439.829,175.155,18.535,152.896
C04936=1089.147,58.692,439.845,175.152,18.533,152.896
C04937=1089.142,58.442,439.862,175.151,18.532,152.896
C04938=1089.137,58.193,439.877,175.149,18.530,152.896
C04939=1089.131,57.944,439.894,175.147,18.529,152.896
C04940=1089.125,57.694,439.910,175.145,18.526,152.896
C04941=1089.119,57.445,439.926,175.143,18.525,152.896
C04942=1089.113,57.196,439.943,175.141,18.523,152.896
C04943=1089.107,56.946,439.959,175.139,18.522,152.896
C04944=1089.102,56.697,439.976,175.138,18.520,152.896
C04945=1089.096,56.447,439.992,175.136,18.519,152.896
C04946=1089.091,56.197,440.007,175.134,18.517,152.896
C04947=1089.085,55.948,440.024,175.132,18.515,152.896
C04948=1089.079,55.699,440.040,175.130,18.514,152.896
C04949=1089.073,55.450,440.056,175.128,18.512,152.896
C04950=1089.067,55.201,440.072,175.127,18.510,152.896
C04951=1089.062,54.951,440.088,175.124,18.508,152.896
C04952=1089.056,54.701,440.104,175.123,18.507,152.896
C04953=1089.051,54.452,440.121,175.120,18.505,152.896
C04954=1089.045,54.202,440.137,175.119,18.504,152.896
C04955=1089.039,53.954,440.153,175.118,18.502,152.896
C04956=1089.034,53.704,440.168,175.115,18.500,152.896
C04957=1089.028,53.454,440.185,175.114,18.499,152.896
C04958=1089.022,53.205,440.201,175.111,18.497,152.896
C04959=1089.016,52.956,440.217,175.110,18.495,152.896
C04960=1089.010,52.706,440.233,175.107,18.494,152.896
C04961=1089.005,52.457,440.249,175.106,18.492,152.896
C04962=1089.000,52.207,440.265,175.104,18.490,152.896
C04963=1088.994,51.957,440.281,175.102,18.488,152.896
C04964=1088.988,51.708,440.297,175.101,18.487,152.896
C04965=1088.982,51.459,440.314,175.098,18.485,152.896
C04966=1088.977,51.209,440.329,175.097,18.484,152.896
C04967=1088.971,50.960,440.345,175.095,18.482,152.896
C04968=1088.965,50.711,440.361,175.093,18.480,152.896
C04969=1088.959,50.461,440.377,175.091,18.479,152.896
C04970=1088.953,50.211,440.393,175.090,18.477,152.896
C04971=1088.948,49.963,440.409,175.088,18.475,152.896
C04972=1088.942,49.713,440.424,175.086,18.473,152.896
C04973=1088.936,49.463,440.441,175.084,18.472,152.896
C04974=1088.931,49.214,440.457,175.082,18.470,152.896
C04975=1088.925,48.965,440.472,175.081,18.469,152.896
C04976=1088.920,48.715,440.488,175.078,18.467,152.896
C04977=1088.914,48.466,440.504,175.077,18.465,152.896
C04978=1088.908,48.216,440.520,175.075,18.463,152.896
C04979=1088.903,47.967,440.535,175.073,18.461,152.896
C04980=1088.897,47.689,440.554,175.071,18.459,152.896
C04981=1088.890,47.413,440.571,175.070,18.458,152.896
C04982=1088.884,47.135,440.589,175.067,18.456,152.896
C04983=1088.877,46.858,440.607,175.065,18.454,152.896
C04984=1088.872,46.608,440.622,175.064,18.452,152.896
C04985=1088.866,46.359,440.638,175.061,18.451,152.896
C04986=1088.861,46.109,440.654,175.060,18.449,152.896
C04987=1088.855,45.860,440.670,175.058,18.447,152.896
C04988=1088.850,45.610,440.685,175.056,18.445,152.896
C04989=1088.844,45.360,440.701,175.055,18.444,152.896
C04990=1088.839,45.112,440.717,175.052,18.442,152.896
C04991=1088.833,44.862,440.732,175.051,18.440,152.896
C04992=1088.827,44.613,440.749,175.049,18.438,152.896
C04993=1088.822,44.363,440.764,175.047,18.436,152.896
C04994=1088.816,44.114,440.780,175.046,18.435,152.896
C04995=1088.811,43.864,440.796,175.044,18.433,152.896
C04996=1088.805,43.615,440.811,175.042,18.432,152.896
C04997=1088.799,43.366,440.826,175.040,18.430,152.896
C04998=1088.793,43.116,440.842,175.038,18.428,152.896
C04999=1088.787,42.866,440.858,175.037,18.427,152.896
C05000=1088.782,42.617,440.873,175.035,18.425,152.896
C05001=1088.776,42.368,440.890,175.033,18.423,152.896
C05002=1088.770,42.118,440.905,175.031,18.421,152.896
C05003=1088.765,41.869,440.920,175.029,18.420,152.896
C05004=1088.759,41.619,440.936,175.028,18.418,152.896
C05005=1088.753,41.369,440.952,175.026,18.416,152.896
C05006=1088.748,41.120,440.967,175.024,18.415,152.896
C05007=1088.741,40.871,440.982,175.022,18.413,152.896
C05008=1088.736,40.621,440.998,175.021,18.411,152.895
C05009=1088.731,40.372,441.013,175.019,18.409,152.895
C05010=1088.725,40.123,441.029,175.017,18.407,152.895
C05011=1088.718,39.873,441.044,175.016,18.406,152.895
C05012=1088.713,39.624,441.059,175.013,18.404,152.896
C05013=1088.707,39.374,441.076,175.012,18.403,152.895
C05014=1088.702,39.125,441.091,175.010,18.401,152.895
C05015=1088.696,38.875,441.106,175.008,18.399,152.895
C05016=1088.690,38.625,441.121,175.007,18.397,152.895
C05017=1088.685,38.377,441.137,175.004,18.395,152.895
C05018=1088.679,38.127,441.153,175.003,18.394,152.895
C05019=1088.673,37.877,441.168,175.002,18.392,152.895
C05020=1088.668,37.628,441.183,174.999,18.390,152.895
C05021=1088.662,37.379,441.199,174.998,18.389,152.895
C05022=1088.656,37.130,441.214,174.996,18.387,152.895
C05023=1088.651,36.880,441.229,174.994,18.385,152.895
C05024=1088.644,36.630,441.244,174.993,18.384,152.895
C05025=1088.639,36.381,441.260,174.990,18.382,152.895
C05026=1088.633,36.131,441.276,174.989,18.380,152.895
C05027=1088.627,35.882,441.291,174.987,18.378,152.895
C05028=1088.622,35.632,441.306,174.985,18.377,152.895
C05029=1088.615,35.383,441.321,174.984,18.375,152.895
C05030=1088.610,35.133,441.336,174.982,18.373,152.895
C05031=1088.604,34.884,441.352,174.980,18.371,152.895
C05032=1088.598,34.634,441.367,174.979,18.370,152.895
C05033=1088.593,34.385,441.382,174.976,18.368,152.895
C05034=1088.587,34.136,441.397,174.975,18.367,152.895
C05035=1088.582,33.886,441.412,174.973,18.365,152.895
C05036=1088.575,33.637,441.427,174.971,18.363,152.895
C05037=1088.570,33.387,441.443,174.970,18.362,152.895
C05038=1088.565,33.137,441.458,174.968,18.359,152.895
C05039=1088.558,32.888,441.473,174.966,18.358,152.895
C05040=1088.553,32.639,441.489,174.965,18.356,152.895
C05041=1088.546,32.389,441.504,174.963,18.354,152.895
C05042=1088.541,32.140,441.519,174.961,18.353,152.895
C05043=1088.535,31.891,441.534,174.959,18.351,152.895
C05044=1088.529,31.613,441.551,174.958,18.349,152.895
C05045=1088.522,31.336,441.568,174.955,18.347,152.895
C05046=1088.516,31.059,441.585,174.953,18.345,152.895
C05047=1088.510,30.781,441.601,174.952,18.343,152.895
C05048=1088.504,30.532,441.616,174.949,18.341,152.895
C05049=1088.499,30.283,441.632,174.948,18.340,152.895
C05050=1088.492,30.033,441.647,174.947,18.338,152.895
C05051=1088.487,29.784,441.662,174.944,18.336,152.895
C05052=1088.481,29.534,441.677,174.943,18.334,152.895
C05053=1088.476,29.285,441.692,174.941,18.333,152.895
C05054=1088.469,29.035,441.707,174.939,18.331,152.895
C05055=1088.465,28.785,441.721,174.938,18.329,152.894
C05056=1088.458,28.535,441.736,174.936,18.328,152.894
C05057=1088.453,28.287,441.751,174.934,18.326,152.894
C05058=1088.447,28.037,441.766,174.933,18.324,152.894
C05059=1088.441,27.788,441.781,174.931,18.323,152.894
C05060=1088.436,27.538,441.796,174.929,18.320,152.894
C05061=1088.430,27.289,441.811,174.928,18.319,152.894
C05062=1088.423,27.039,441.826,174.926,18.317,152.894
C05063=1088.418,26.790,441.841,174.924,18.315,152.894
C05064=1088.412,26.540,441.856,174.923,18.314,152.894
C05065=1088.406,26.291,441.871,174.920,18.312,152.894
C05066=1088.401,26.041,441.885,174.919,18.310,152.894
C05067=1088.395,25.792,441.900,174.918,18.308,152.894
C05068=1088.389,25.542,441.915,174.915,18.306,152.894
C05069=1088.384,25.293,441.930,174.914,18.305,152.894
C05070=1088.377,25.043,441.945,174.913,18.303,152.894
C05071=1088.371,24.794,441.960,174.910,18.301,152.894
C05072=1088.366,24.543,441.975,174.909,18.300,152.894
C05073=1088.360,24.295,441.989,174.908,18.298,152.894
C05074=1088.354,24.045,442.004,174.905,18.296,152.894
C05075=1088.349,23.796,442.019,174.904,18.294,152.894
C05076=1088.342,23.546,442.034,174.902,18.293,152.894
C05077=1088.337,23.296,442.048,174.900,18.291,152.894
C05078=1088.331,23.046,442.064,174.899,18.289,152.894
C05079=1088.326,22.797,442.078,174.897,18.288,152.894
C05080=1088.320,22.548,442.093,174.895,18.286,152.894
C05081=1088.313,22.299,442.108,174.894,18.284,152.894
C05082=1088.309,22.049,442.122,174.892,18.282,152.894
C05083=1088.302,21.799,442.137,174.890,18.280,152.894
C05084=1088.297,21.550,442.152,174.889,18.279,152.894
C05085=1088.291,21.300,442.166,174.887,18.277,152.893
C05086=1088.285,21.051,442.181,174.885,18.275,152.893
C05087=1088.280,20.802,442.196,174.884,18.274,152.893
C05088=1088.273,20.552,442.211,174.882,18.272,152.893
C05089=1088.269,20.302,442.225,174.880,18.270,152.893
C05090=1088.262,20.053,442.240,174.879,18.268,152.893
C05091=1088.256,19.804,442.255,174.877,18.267,152.893
C05092=1088.251,19.554,442.268,174.875,18.265,152.893
C05093=1088.244,19.304,442.283,174.874,18.263,152.893
C05094=1088.239,19.055,442.298,174.872,18.262,152.893
C05095=1088.233,18.805,442.313,174.870,18.259,152.893
C05096=1088.228,18.556,442.327,174.869,18.258,152.893
C05097=1088.222,18.306,442.341,174.867,18.256,152.893
C05098=1088.216,18.057,442.356,174.865,18.254,152.893
C05099=1088.210,17.808,442.371,174.863,18.253,152.893
C05100=1088.204,17.557,442.385,174.862,18.251,152.893
C05101=1088.199,17.308,442.400,174.860,18.249,152.893
C05102=1088.193,17.059,442.414,174.858,18.248,152.893
C05103=1088.187,16.809,442.429,174.857,18.246,152.893
C05104=1088.181,16.560,442.444,174.855,18.244,152.893
C05105=1088.176,16.310,442.457,174.853,18.242,152.893
C05106=1088.169,16.061,442.472,174.852,18.241,152.893
C05107=1088.164,15.811,442.486,174.850,18.239,152.893
C05108=1088.157,15.536,442.503,174.848,18.237,152.893
C05109=1088.151,15.260,442.519,174.846,18.234,152.893
C05110=1088.145,14.984,442.534,174.845,18.233,152.893
C05111=1088.139,14.708,442.550,174.843,18.231,152.893
C05112=1088.133,14.459,442.565,174.841,18.229,152.892
C05113=1088.127,14.208,442.579,174.839,18.227,152.892
C05114=1088.121,13.959,442.594,174.838,18.226,152.892
C05115=1088.115,13.709,442.608,174.836,18.224,152.892
C05116=1088.109,13.460,442.622,174.835,18.222,152.892
C05117=1088.104,13.211,442.636,174.833,18.220,152.892
C05118=1088.097,12.961,442.651,174.831,18.219,152.892
C05119=1088.092,12.711,442.665,174.830,18.217,152.892
C05120=1088.086,12.462,442.680,174.828,18.215,152.892
C05121=1088.080,12.212,442.694,174.826,18.214,152.892
C05122=1088.074,11.963,442.709,174.825,18.212,152.892
C05123=1088.069,11.714,442.722,174.823,18.210,152.892
C05124=1088.062,11.464,442.736,174.821,18.208,152.892
C05125=1088.056,11.215,442.751,174.820,18.207,152.892
C05126=1088.051,10.965,442.764,174.818,18.205,152.892
C05127=1088.044,10.715,442.779,174.816,18.203,152.892
C05128=1088.039,10.466,442.793,174.815,18.202,152.892
C05129=1088.033,10.216,442.807,174.813,18.200,152.892
C05130=1088.027,9.967,442.822,174.811,18.198,152.892
C05131=1088.022,9.717,442.836,174.810,18.196,152.892
C05132=1088.016,9.467,442.850,174.808,18.195,152.892
C05133=1088.010,9.218,442.865,174.806,18.193,152.892
C05134=1088.004,8.968,442.879,174.805,18.191,152.892
C05135=1087.998,8.719,442.892,174.803,18.190,152.892
C05136=1087.992,8.470,442.906,174.802,18.188,152.892
C05137=1087.986,8.220,442.921,174.800,18.186,152.892
C05138=1087.981,7.970,442.935,174.798,18.184,152.892
C05139=1087.975,7.721,442.949,174.797,18.183,152.892
C05140=1087.969,7.471,442.963,174.795,18.181,152.892
C05141=1087.963,7.221,442.977,174.793,18.179,152.892
C05142=1087.958,6.972,442.992,174.792,18.178,152.891
C05143=1087.951,6.723,443.005,174.790,18.176,152.891
C05144=1087.945,6.473,443.019,174.788,18.174,152.891
C05145=1087.940,6.223,443.033,174.787,18.172,152.891
C05146=1087.934,5.974,443.048,174.786,18.170,152.891
C05147=1087.929,5.725,443.062,174.783,18.168,152.891
C05148=1087.923,5.475,443.075,174.782,18.167,152.891
C05149=1087.917,5.225,443.090,174.781,18.165,152.891
C05150=1087.910,4.976,443.104,174.779,18.164,152.891
C05151=1087.905,4.727,443.118,174.777,18.161,152.891
C05152=1087.899,4.477,443.131,174.775,18.160,152.891
C05153=1087.893,4.227,443.146,174.774,18.158,152.891
C05154=1087.888,3.977,443.160,174.772,18.156,152.891
C05155=1087.882,3.728,443.173,174.770,18.155,152.891
C05156=1087.876,3.479,443.187,174.769,18.153,152.891
C05157=1087.870,3.229,443.201,174.768,18.152,152.891
C05158=1087.865,2.980,443.215,174.765,18.149,152.891
C05159=1087.859,2.730,443.229,174.764,18.148,152.891
C05160=1087.853,2.480,443.243,174.763,18.146,152.891
C05161=1087.847,2.231,443.256,174.761,18.144,152.891
C05162=1087.841,1.982,443.271,174.759,18.142,152.891
C05163=1087.836,1.732,443.285,174.758,18.141,152.891
C05164=1087.830,1.483,443.299,174.756,18.139,152.890
C05165=1087.824,1.232,443.313,174.754,18.137,152.890
C05166=1087.818,0.983,443.326,174.753,18.135,152.890
C05167=1087.813,0.734,443.340,174.751,18.134,152.890
C05168=1087.807,0.484,443.354,174.750,18.132,152.890
C05169=1087.802,0.234,443.368,174.748,18.130,152.890
C05170=1087.796,-0.015,443.381,174.746,18.129,152.890
C05171=1087.790,-0.264,443.395,174.745,18.126,152.890
C05172=1087.783,-0.539,443.411,174.743,18.124,152.890
C05173=1087.777,-0.813,443.426,174.742,18.123,152.890
C05174=1087.771,-1.086,443.441,174.739,18.121,152.890
C05175=1087.765,-1.360,443.456,174.738,18.119,152.890
C05176=1087.759,-1.610,443.470,174.737,18.117,152.890
C05177=1087.753,-1.859,443.484,174.735,18.115,152.890
C05178=1087.748,-2.109,443.498,174.733,18.113,152.890
C05179=1087.742,-2.359,443.511,174.732,18.112,152.890
C05180=1087.736,-2.608,443.525,174.730,18.110,152.890
C05181=1087.730,-2.857,443.539,174.728,18.108,152.890
C05182=1087.725,-3.107,443.552,174.727,18.107,152.890
C05183=1087.719,-3.356,443.566,174.725,18.105,152.890
C05184=1087.713,-3.606,443.580,174.723,18.103,152.890
C05185=1087.708,-3.855,443.593,174.722,18.101,152.890
C05186=1087.701,-4.105,443.607,174.720,18.100,152.889
C05187=1087.695,-4.355,443.621,174.719,18.098,152.889
C05188=1087.690,-4.605,443.633,174.717,18.096,152.889
C05189=1087.684,-4.854,443.647,174.715,18.095,152.889
C05190=1087.678,-5.104,443.661,174.714,18.093,152.889
C05191=1087.672,-5.353,443.674,174.713,18.091,152.889
C05192=1087.666,-5.603,443.688,174.711,18.089,152.889
C05193=1087.661,-5.852,443.702,174.709,18.087,152.889
C05194=1087.654,-6.102,443.715,174.708,18.086,152.889
C05195=1087.648,-6.352,443.729,174.706,18.084,152.889
C05196=1087.642,-6.601,443.742,174.704,18.082,152.889
C05197=1087.637,-6.850,443.756,174.703,18.080,152.889
C05198=1087.631,-7.100,443.769,174.701,18.079,152.889
C05199=1087.625,-7.350,443.783,174.700,18.077,152.889
C05200=1087.619,-7.599,443.796,174.698,18.076,152.889
C05201=1087.614,-7.849,443.810,174.696,18.074,152.889
C05202=1087.607,-8.098,443.823,174.695,18.072,152.889
C05203=1087.602,-8.348,443.837,174.693,18.071,152.889
C05204=1087.596,-8.598,443.849,174.692,18.069,152.889
C05205=1087.591,-8.847,443.863,174.690,18.067,152.889
C05206=1087.584,-9.096,443.877,174.688,18.065,152.889
C05207=1087.578,-9.347,443.891,174.687,18.064,152.889
C05208=1087.572,-9.596,443.904,174.686,18.062,152.889
C05209=1087.567,-9.846,443.917,174.683,18.060,152.889
C05210=1087.561,-10.095,443.931,174.682,18.059,152.889
C05211=1087.554,-10.345,443.944,174.681,18.057,152.888
C05212=1087.549,-10.594,443.958,174.679,18.055,152.888
C05213=1087.543,-10.844,443.970,174.677,18.053,152.888
C05214=1087.538,-11.094,443.984,174.676,18.052,152.888
C05215=1087.531,-11.343,443.997,174.674,18.050,152.888
C05216=1087.526,-11.592,444.011,174.673,18.048,152.888
C05217=1087.520,-11.842,444.024,174.672,18.047,152.888
C05218=1087.515,-12.092,444.038,174.669,18.044,152.888
C05219=1087.508,-12.341,444.051,174.668,18.043,152.888
C05220=1087.502,-12.591,444.063,174.667,18.041,152.888
C05221=1087.497,-12.841,444.077,174.665,18.040,152.888
C05222=1087.491,-13.090,444.091,174.663,18.038,152.888
C05223=1087.486,-13.340,444.104,174.662,18.036,152.888
C05224=1087.479,-13.589,444.117,174.660,18.034,152.888
C05225=1087.474,-13.839,444.131,174.659,18.033,152.888
C05226=1087.468,-14.089,444.143,174.657,18.031,152.888
C05227=1087.462,-14.338,444.157,174.655,18.029,152.888
C05228=1087.456,-14.588,444.171,174.654,18.028,152.888
C05229=1087.451,-14.837,444.183,174.652,18.026,152.888
C05230=1087.445,-15.086,444.197,174.651,18.025,152.888
C05231=1087.440,-15.336,444.209,174.649,18.022,152.888
C05232=1087.433,-15.586,444.222,174.647,18.021,152.888
C05233=1087.427,-15.835,444.236,174.646,18.019,152.888
C05234=1087.422,-16.085,444.249,174.645,18.018,152.888
C05235=1087.416,-16.334,444.262,174.643,18.016,152.887
C05236=1087.409,-16.607,444.276,174.641,18.014,152.888
C05237=1087.402,-16.879,444.291,174.640,18.012,152.887
C05238=1087.396,-17.151,444.305,174.638,18.010,152.887
C05239=1087.390,-17.424,444.319,174.636,18.008,152.887
C05240=1087.384,-17.673,444.333,174.635,18.007,152.887
C05241=1087.378,-17.923,444.345,174.633,18.005,152.887
C05242=1087.372,-18.172,444.358,174.631,18.003,152.887
C05243=1087.365,-18.422,444.372,174.630,18.001,152.887
C05244=1087.360,-18.672,444.385,174.628,18.000,152.887
C05245=1087.354,-18.921,444.398,174.627,17.998,152.887
C05246=1087.348,-19.171,444.411,174.626,17.997,152.887
C05247=1087.343,-19.420,444.423,174.623,17.995,152.887
C05248=1087.337,-19.669,444.436,174.622,17.993,152.887
C05249=1087.331,-19.919,444.450,174.621,17.992,152.887
C05250=1087.325,-20.169,444.462,174.619,17.990,152.887
C05251=1087.319,-20.419,444.475,174.618,17.988,152.887
C05252=1087.313,-20.668,444.488,174.616,17.986,152.887
C05253=1087.307,-20.918,444.501,174.614,17.985,152.887
C05254=1087.302,-21.168,444.515,174.613,17.983,152.887
C05255=1087.296,-21.417,444.527,174.611,17.982,152.887
C05256=1087.290,-21.667,444.541,174.610,17.980,152.887
C05257=1087.284,-21.917,444.553,174.608,17.978,152.887
C05258=1087.277,-22.166,444.566,174.606,17.976,152.887
C05259=1087.272,-22.415,444.579,174.605,17.975,152.887
C05260=1087.267,-22.665,444.592,174.604,17.973,152.887
C05261=1087.261,-22.914,444.605,174.602,17.972,152.886
C05262=1087.255,-23.164,444.618,174.600,17.970,152.887
C05263=1087.249,-23.414,444.630,174.599,17.968,152.886
C05264=1087.243,-23.664,444.643,174.597,17.966,152.886
C05265=1087.237,-23.913,444.656,174.596,17.965,152.886
C05266=1087.232,-24.162,444.669,174.594,17.963,152.886
C05267=1087.226,-24.412,444.682,174.592,17.961,152.886
C05268=1087.220,-24.662,444.694,174.591,17.960,152.886
C05269=1087.214,-24.911,444.708,174.589,17.958,152.886
C05270=1087.208,-25.161,444.720,174.588,17.956,152.886
C05271=1087.202,-25.411,444.733,174.587,17.955,152.886
C05272=1087.196,-25.660,444.746,174.585,17.953,152.886
C05273=1087.191,-25.910,444.758,174.583,17.951,152.886
C05274=1087.185,-26.160,444.771,174.581,17.950,152.886
C05275=1087.180,-26.410,444.784,174.580,17.948,152.886
C05276=1087.173,-26.659,444.797,174.579,17.946,152.886
C05277=1087.167,-26.909,444.810,174.577,17.945,152.886
C05278=1087.162,-27.158,444.822,174.575,17.943,152.886
C05279=1087.156,-27.407,444.835,174.574,17.941,152.886
C05280=1087.150,-27.657,444.848,174.572,17.940,152.886
C05281=1087.144,-27.907,444.860,174.571,17.938,152.886
C05282=1087.138,-28.157,444.873,174.570,17.937,152.886
C05283=1087.132,-28.406,444.886,174.568,17.935,152.886
C05284=1087.126,-28.656,444.899,174.566,17.933,152.886
C05285=1087.120,-28.905,444.910,174.564,17.932,152.886
C05286=1087.114,-29.155,444.923,174.563,17.930,152.886
C05287=1087.108,-29.405,444.935,174.561,17.929,152.886
C05288=1087.102,-29.654,444.949,174.560,17.927,152.886
C05289=1087.096,-29.904,444.961,174.559,17.925,152.886
C05290=1087.090,-30.154,444.974,174.557,17.924,152.886
C05291=1087.085,-30.403,444.986,174.555,17.922,152.886
C05292=1087.079,-30.653,444.999,174.554,17.920,152.886
C05293=1087.073,-30.902,445.012,174.552,17.919,152.886
C05294=1087.067,-31.152,445.024,174.551,17.917,152.886
C05295=1087.061,-31.402,445.037,174.549,17.916,152.885
C05296=1087.056,-31.651,445.049,174.548,17.914,152.885
C05297=1087.049,-31.901,445.061,174.546,17.912,152.886
C05298=1087.043,-32.150,445.074,174.544,17.911,152.886
C05299=1087.037,-32.400,445.086,174.543,17.909,152.885
C05300=1087.030,-32.671,445.100,174.541,17.908,152.885
C05301=1087.024,-32.943,445.114,174.539,17.906,152.885
C05302=1087.018,-33.215,445.127,174.538,17.904,152.885
C05303=1087.011,-33.486,445.141,174.536,17.902,152.885
C05304=1087.006,-33.735,445.153,174.535,17.901,152.885
C05305=1087.000,-33.985,445.166,174.533,17.899,152.885
C05306=1086.994,-34.235,445.178,174.531,17.897,152.885
C05307=1086.988,-34.484,445.191,174.530,17.896,152.885
C05308=1086.983,-34.734,445.203,174.529,17.894,152.885
C05309=1086.977,-34.983,445.215,174.527,17.892,152.885
C05310=1086.971,-35.233,445.228,174.526,17.891,152.885
C05311=1086.964,-35.483,445.240,174.524,17.889,152.885
C05312=1086.959,-35.732,445.252,174.522,17.887,152.885
C05313=1086.953,-35.982,445.265,174.521,17.886,152.885
C05314=1086.947,-36.232,445.277,174.519,17.884,152.885
C05315=1086.941,-36.482,445.290,174.518,17.883,152.885
C05316=1086.936,-36.731,445.302,174.516,17.881,152.885
C05317=1086.929,-36.981,445.314,174.515,17.880,152.885
C05318=1086.924,-37.230,445.326,174.514,17.878,152.885
C05319=1086.918,-37.480,445.339,174.511,17.876,152.885
C05320=1086.912,-37.729,445.351,174.510,17.875,152.885
C05321=1086.906,-37.979,445.364,174.509,17.873,152.885
C05322=1086.901,-38.229,445.376,174.507,17.871,152.885
C05323=1086.894,-38.478,445.388,174.506,17.870,152.885
C05324=1086.889,-38.728,445.400,174.504,17.868,152.885
C05325=1086.883,-38.977,445.413,174.503,17.867,152.885
C05326=1086.877,-39.227,445.425,174.501,17.866,152.885
C05327=1086.871,-39.477,445.437,174.499,17.864,152.885
C05328=1086.865,-39.727,445.450,174.498,17.862,152.885
C05329=1086.859,-39.976,445.462,174.496,17.860,152.885
C05330=1086.853,-40.225,445.474,174.495,17.859,152.885
C05331=1086.847,-40.475,445.486,174.494,17.857,152.885
C05332=1086.842,-40.725,445.498,174.492,17.856,152.885
C05333=1086.835,-40.975,445.510,174.490,17.855,152.885
C05334=1086.829,-41.224,445.522,174.489,17.853,152.885
C05335=1086.823,-41.474,445.534,174.488,17.851,152.885
C05336=1086.817,-41.723,445.547,174.485,17.849,152.885
C05337=1086.811,-41.973,445.559,174.484,17.848,152.885
C05338=1086.805,-42.223,445.571,174.482,17.847,152.885
C05339=1086.800,-42.472,445.583,174.481,17.845,152.885
C05340=1086.794,-42.722,445.595,174.480,17.844,152.885
C05341=1086.787,-42.972,445.607,174.478,17.842,152.885
C05342=1086.782,-43.221,445.619,174.477,17.840,152.885
C05343=1086.776,-43.471,445.632,174.475,17.839,152.885
C05344=1086.769,-43.721,445.644,174.474,17.838,152.885
C05345=1086.764,-43.970,445.655,174.472,17.836,152.885
C05346=1086.758,-44.220,445.667,174.470,17.834,152.885
C05347=1086.752,-44.470,445.680,174.469,17.833,152.885
C05348=1086.747,-44.719,445.692,174.467,17.831,152.885
C05349=1086.740,-44.969,445.704,174.466,17.830,152.885
C05350=1086.735,-45.218,445.715,174.464,17.828,152.885
C05351=1086.728,-45.468,445.727,174.463,17.827,152.885
C05352=1086.722,-45.718,445.740,174.462,17.825,152.884
C05353=1086.717,-45.967,445.752,174.460,17.824,152.884
C05354=1086.711,-46.217,445.763,174.458,17.822,152.885
C05355=1086.705,-46.466,445.775,174.456,17.820,152.885
C05356=1086.699,-46.716,445.787,174.455,17.819,152.885
C05357=1086.693,-46.966,445.800,174.453,17.817,152.884
C05358=1086.687,-47.215,445.811,174.452,17.816,152.884
C05359=1086.681,-47.465,445.823,174.451,17.814,152.884
C05360=1086.676,-47.714,445.836,174.449,17.813,152.885
C05361=1086.670,-47.965,445.847,174.448,17.811,152.884
C05362=1086.664,-48.214,445.859,174.446,17.810,152.884
C05363=1086.658,-48.463,445.871,174.445,17.808,152.884
C05364=1086.652,-48.736,445.884,174.443,17.806,152.884
C05365=1086.645,-49.007,445.897,174.441,17.805,152.884
C05366=1086.639,-49.279,445.910,174.440,17.804,152.884
C05367=1086.632,-49.551,445.922,174.438,17.802,152.884
C05368=1086.626,-49.801,445.935,174.436,17.800,152.884
C05369=1086.620,-50.050,445.946,174.435,17.798,152.884
C05370=1086.615,-50.300,445.958,174.433,17.797,152.884
C05371=1086.609,-50.549,445.970,174.432,17.796,152.884
C05372=1086.603,-50.799,445.982,174.430,17.794,152.884
C05373=1086.596,-51.049,445.994,174.429,17.793,152.884
C05374=1086.590,-51.298,446.005,174.427,17.791,152.884
C05375=1086.585,-51.548,446.017,174.426,17.790,152.884
C05376=1086.578,-51.798,446.029,174.424,17.788,152.884
C05377=1086.572,-52.047,446.040,174.423,17.787,152.885
C05378=1086.566,-52.297,446.052,174.421,17.786,152.884
C05379=1086.560,-52.546,446.064,174.420,17.784,152.884
C05380=1086.554,-52.796,446.075,174.418,17.783,152.885
C05381=1086.548,-53.046,446.088,174.417,17.781,152.884
C05382=1086.542,-53.296,446.099,174.415,17.780,152.884
C05383=1086.536,-53.545,446.111,174.413,17.778,152.885
C05384=1086.530,-53.795,446.121,174.412,17.777,152.885
C05385=1086.524,-54.045,446.134,174.410,17.775,152.885
C05386=1086.517,-54.294,446.146,174.409,17.774,152.885
C05387=1086.512,-54.544,446.157,174.407,17.772,152.885
C05388=1086.506,-54.794,446.169,174.406,17.771,152.885
C05389=1086.500,-55.043,446.180,174.404,17.770,152.885
C05390=1086.493,-55.293,446.192,174.403,17.768,152.885
C05391=1086.488,-55.542,446.203,174.401,17.767,152.885
C05392=1086.482,-55.792,446.216,174.400,17.766,152.885
C05393=1086.476,-56.042,446.227,174.398,17.764,152.885
C05394=1086.470,-56.292,446.238,174.397,17.762,152.885
C05395=1086.463,-56.541,446.250,174.395,17.761,152.885
C05396=1086.458,-56.791,446.261,174.394,17.760,152.885
C05397=1086.451,-57.041,446.273,174.392,17.759,152.885
C05398=1086.446,-57.290,446.284,174.391,17.757,152.885
C05399=1086.439,-57.540,446.296,174.389,17.756,152.885
C05400=1086.434,-57.790,446.307,174.388,17.755,152.885
C05401=1086.427,-58.039,446.319,174.386,17.753,152.885
C05402=1086.422,-58.289,446.330,174.384,17.751,152.885
C05403=1086.415,-58.539,446.342,174.382,17.750,152.885
C05404=1086.409,-58.788,446.353,174.381,17.748,152.885
C05405=1086.404,-59.038,446.365,174.380,17.747,152.885
C05406=1086.398,-59.287,446.377,174.378,17.746,152.885
C05407=1086.391,-59.537,446.388,174.377,17.744,152.885
C05408=1086.385,-59.787,446.399,174.375,17.743,152.885
C05409=1086.380,-60.037,446.411,174.374,17.741,152.885
C05410=1086.374,-60.286,446.422,174.372,17.740,152.885
C05411=1086.368,-60.536,446.433,174.371,17.739,152.885
C05412=1086.361,-60.785,446.445,174.369,17.737,152.885
C05413=1086.356,-61.035,446.456,174.368,17.736,152.885
C05414=1086.349,-61.285,446.467,174.366,17.735,152.885
C05415=1086.344,-61.534,446.479,174.365,17.733,152.885
C05416=1086.338,-61.784,446.491,174.363,17.732,152.885
C05417=1086.332,-62.034,446.501,174.362,17.730,152.885
C05418=1086.325,-62.283,446.513,174.360,17.729,152.885
C05419=1086.320,-62.533,446.524,174.359,17.728,152.885
C05420=1086.314,-62.783,446.536,174.357,17.726,152.885
C05421=1086.308,-63.032,446.548,174.356,17.725,152.885
C05422=1086.302,-63.282,446.559,174.354,17.723,152.885
C05423=1086.296,-63.532,446.570,174.353,17.722,152.885
C05424=1086.290,-63.781,446.581,174.351,17.721,152.885
C05425=1086.283,-64.031,446.593,174.350,17.719,152.885
C05426=1086.278,-64.281,446.604,174.348,17.718,152.885
C05427=1086.272,-64.531,446.615,174.347,17.717,152.885
C05428=1086.265,-64.803,446.627,174.345,17.715,152.885
C05429=1086.259,-65.076,446.640,174.343,17.713,152.885
C05430=1086.252,-65.349,446.652,174.341,17.712,152.885
C05431=1086.246,-65.623,446.665,174.340,17.711,152.885
C05432=1086.240,-65.873,446.676,174.338,17.709,152.885
C05433=1086.235,-66.122,446.686,174.337,17.708,152.885
C05434=1086.228,-66.372,446.698,174.335,17.707,152.886
C05435=1086.222,-66.621,446.709,174.334,17.705,152.885
C05436=1086.216,-66.871,446.721,174.332,17.704,152.886
C05437=1086.211,-67.121,446.732,174.331,17.702,152.886
C05438=1086.205,-67.371,446.743,174.329,17.701,152.886
C05439=1086.199,-67.621,446.754,174.328,17.700,152.886
C05440=1086.193,-67.870,446.766,174.327,17.698,152.886
C05441=1086.187,-68.119,446.777,174.325,17.697,152.886
C05442=1086.181,-68.369,446.788,174.323,17.695,152.886
C05443=1086.175,-68.619,446.799,174.322,17.694,152.886
C05444=1086.169,-68.868,446.810,174.320,17.693,152.886
C05445=1086.163,-69.118,446.821,174.319,17.692,152.886
C05446=1086.158,-69.368,446.832,174.317,17.690,152.886
C05447=1086.152,-69.618,446.843,174.316,17.689,152.886
C05448=1086.146,-69.867,446.855,174.314,17.688,152.886
C05449=1086.140,-70.117,446.866,174.313,17.686,152.886
C05450=1086.134,-70.366,446.877,174.311,17.685,152.886
C05451=1086.128,-70.617,446.888,174.310,17.683,152.886
C05452=1086.122,-70.866,446.899,174.308,17.682,152.886
C05453=1086.116,-71.115,446.910,174.307,17.681,152.886
C05454=1086.111,-71.365,446.921,174.305,17.680,152.886
C05455=1086.104,-71.615,446.932,174.304,17.678,152.886
C05456=1086.098,-71.865,446.943,174.302,17.677,152.886
C05457=1086.093,-72.114,446.954,174.301,17.675,152.886
C05458=1086.086,-72.364,446.965,174.299,17.674,152.886
C05459=1086.081,-72.614,446.976,174.298,17.673,152.886
C05460=1086.076,-72.864,446.987,174.296,17.672,152.886
C05461=1086.070,-73.113,446.998,174.295,17.670,152.886
C05462=1086.064,-73.363,447.009,174.293,17.669,152.886
C05463=1086.058,-73.613,447.020,174.292,17.667,152.886
C05464=1086.052,-73.862,447.031,174.290,17.666,152.886
C05465=1086.046,-74.112,447.042,174.289,17.665,152.886
C05466=1086.040,-74.362,447.053,174.287,17.664,152.887
